// TIA Portal V16 program export: 1 tag tables, 16 data types, 7 data blocks, 22 code blocks (in call order from the OBs), 5 instance data blocks

VAR_GLOBAL   // PLC tag table "Default tag table"
   System_Byte AT %MB1 : Byte;
   FirstScan AT %M1.0 : Bool;
   DiagStatusUpdate AT %M1.1 : Bool;
   AlwaysTRUE AT %M1.2 : Bool;
   AlwaysFALSE AT %M1.3 : Bool;
   Clock_Byte AT %MB0 : Byte;
   Clock_10Hz AT %M0.0 : Bool;
   Clock_5Hz AT %M0.1 : Bool;
   "Clock_2.5Hz" AT %M0.2 : Bool;
   Clock_2Hz AT %M0.3 : Bool;
   "Clock_1.25Hz" AT %M0.4 : Bool;
   Clock_1Hz AT %M0.5 : Bool;
   "Clock_0.625Hz" AT %M0.6 : Bool;
   "Clock_0.5Hz" AT %M0.7 : Bool;
   ala AT %MW2 : Int;
   "di24.2" AT %I0.2 : Bool;
   diSAFETY AT %I0.3 : Bool;
   diC201FC01 AT %I0.4 : Bool;
   diC202FC01 AT %I0.5 : Bool;
   diC202AV03c AT %I0.6 : Bool;
   diC202AV04c AT %I0.7 : Bool;
   diC201AV01c AT %I1.0 : Bool;
   diC201AV02c AT %I1.1 : Bool;
   diC202AV01c AT %I1.2 : Bool;
   diC202AV02c AT %I1.3 : Bool;
   diC211AV01c AT %I1.4 : Bool;
   diC212AV01c AT %I1.5 : Bool;
   diC2A1AV01c AT %I1.6 : Bool;
   diC2A1AV02c AT %I1.7 : Bool;
   diC2A1AV11c AT %I2.0 : Bool;
   diC2A1AV12c AT %I2.1 : Bool;
   diC2A1AV31c AT %I2.2 : Bool;
   diC2A1AV41c AT %I2.3 : Bool;
   diC2D1AV01c AT %I2.4 : Bool;
   diC2D1AV11c AT %I2.5 : Bool;
   diC2D1AV41c AT %I2.6 : Bool;
   diC2D1AV42c AT %I2.7 : Bool;
   diC2D2AV01c AT %I3.0 : Bool;
   diC2D2AV11c AT %I3.1 : Bool;
   diC2D2AV41c AT %I3.2 : Bool;
   diC2D2AV42c AT %I3.3 : Bool;
   diC2D3AV01c AT %I3.4 : Bool;
   diC2D3AV11c AT %I3.5 : Bool;
   diC2D3AV31c AT %I3.6 : Bool;
   diC2D3AV41c AT %I3.7 : Bool;
   diC2D3AV42c AT %I4.0 : Bool;
   diC2D3AV43c AT %I4.1 : Bool;
   diC2L1AV01c AT %I4.2 : Bool;
   diC2L1AV02c AT %I4.3 : Bool;
   diC2L1AV11c AT %I4.4 : Bool;
   diC2L1AV12c AT %I4.5 : Bool;
   diC2L1AV31c AT %I4.6 : Bool;
   diC2L1AV41c AT %I4.7 : Bool;
   diC2R1AV01c AT %I5.0 : Bool;
   diC2R1AV02c AT %I5.1 : Bool;
   diC2R1AV11c AT %I5.2 : Bool;
   diC2R1AV12c AT %I5.3 : Bool;
   diC2R1AV41c AT %I5.4 : Bool;
   diC2W1AV02c AT %I5.5 : Bool;
   diC2W1AV31c AT %I5.6 : Bool;
   diC2W1AV41c AT %I5.7 : Bool;
   diC211FV01 AT %I6.0 : Bool;
   diC212FV01 AT %I6.1 : Bool;
   diC2D1FV81 AT %I6.2 : Bool;
   diC2D2FV81 AT %I6.3 : Bool;
   diC2A1PD01 AT %I6.4 : Bool;
   diC2D1PD01 AT %I6.5 : Bool;
   diC2D2PD01 AT %I6.6 : Bool;
   diC2D3PD01 AT %I6.7 : Bool;
   diC2L1PD01 AT %I7.0 : Bool;
   diC2R1PD01 AT %I7.1 : Bool;
   diC2W1PD01 AT %I7.2 : Bool;
   diC2A1LL01 AT %I7.3 : Bool;
   diC2D1LL01 AT %I7.4 : Bool;
   diC2D2LL01 AT %I7.5 : Bool;
   diC2D3LL01 AT %I7.6 : Bool;
   diC2L1LL01 AT %I7.7 : Bool;
   diC2R1LL01 AT %I8.0 : Bool;
   diC2W1LL01 AT %I8.1 : Bool;
   diC2A1LH01 AT %I8.2 : Bool;
   diC2D1LH01 AT %I8.3 : Bool;
   diC2D2LH01 AT %I8.4 : Bool;
   diC2D3LH01 AT %I8.5 : Bool;
   diC2L1LH01 AT %I8.6 : Bool;
   diC2R1LH01 AT %I8.7 : Bool;
   diC2W1LH01 AT %I9.0 : Bool;
   doC201AV21b AT %Q0.0 : Bool;
   doC202AV21b AT %Q0.1 : Bool;
   doC2W1AV31b AT %Q0.2 : Bool;
   doC2W1AV02b AT %Q0.3 : Bool;
   doC2R1AV11b AT %Q0.4 : Bool;
   doC2R1AV12b AT %Q0.5 : Bool;
   doC2R1AV41b AT %Q0.6 : Bool;
   doC2R1AV01b AT %Q0.7 : Bool;
   doC2R1AV02b AT %Q1.0 : Bool;
   doC2L1AV11b AT %Q1.1 : Bool;
   doC2L1AV12b AT %Q1.2 : Bool;
   doC2L1AV41b AT %Q1.3 : Bool;
   doC2L1AV01b AT %Q1.4 : Bool;
   doC2L1AV02b AT %Q1.5 : Bool;
   doC2L1AV31b AT %Q1.6 : Bool;
   doC2A1AV11b AT %Q1.7 : Bool;
   doC2A1AV12b AT %Q2.0 : Bool;
   doC2A1AV41b AT %Q2.1 : Bool;
   doC2A1AV01b AT %Q2.2 : Bool;
   doC2A1AV02b AT %Q2.3 : Bool;
   doC2A1AV31b AT %Q2.4 : Bool;
   doC2D1AV11b AT %Q2.5 : Bool;
   doC2D1AV41b AT %Q2.6 : Bool;
   doC2D1AV42b AT %Q2.7 : Bool;
   doC2D1AV01b AT %Q3.0 : Bool;
   doC2D2AV01b AT %Q3.1 : Bool;
   doC2D2AV42b AT %Q3.2 : Bool;
   doC2D2AV41b AT %Q3.3 : Bool;
   doC2D2AV11b AT %Q3.4 : Bool;
   doC2D3AV41b AT %Q3.5 : Bool;
   doC2D3AV42b AT %Q3.6 : Bool;
   doC2D3AV11b AT %Q3.7 : Bool;
   doC2D3AV31b AT %Q4.0 : Bool;
   doC2D3AV43b AT %Q4.1 : Bool;
   doC2D3AV01b AT %Q4.2 : Bool;
   doC202AV01b AT %Q4.3 : Bool;
   doC202AV02b AT %Q4.4 : Bool;
   doC201AV01b AT %Q4.5 : Bool;
   doC201AV02b AT %Q4.6 : Bool;
   doC2A1AV42b AT %Q5.0 : Bool;
   doC2L1AV42b AT %Q5.1 : Bool;
   doC2D1AV81b AT %Q5.3 : Bool;
   doC2D2AV81b AT %Q5.4 : Bool;
   doC2W1AV41b AT %Q5.5 : Bool;
   doC211AV01b AT %Q5.6 : Bool;
   doC212AV01b AT %Q5.7 : Bool;
   doC202AV03b AT %Q6.0 : Bool;
   doC202AV04b AT %Q6.1 : Bool;
   doC2A1MP41b AT %Q6.6 : Bool;
   doC2L1MP41b AT %Q6.7 : Bool;
   doBuczek AT %Q7.0 : Bool;
   doZielona AT %Q7.1 : Bool;
   doCzerwona AT %Q7.2 : Bool;
   doZolta AT %Q7.3 : Bool;
   aiC2W1TT01 AT %IW10 : Int;
   aiC2R1TT01 AT %IW12 : Int;
   aiC2L1TT01 AT %IW14 : Int;
   aiC2A1TT01 AT %IW16 : Int;
   aiC2D1TT01 AT %IW18 : Int;
   aiC2D2TT01 AT %IW20 : Int;
   aiC2D3TT01 AT %IW22 : Int;
   aiC211TT01 AT %IW24 : Int;
   aiC212TT01 AT %IW26 : Int;
   aiC201TT01 AT %IW28 : Int;
   aiC202TT01 AT %IW30 : Int;
   aiC212QIC01 AT %IW32 : Int;
   aiC211QIC01 AT %IW34 : Int;
   aiC2A1LT01 AT %IW36 : Int;
   aiC2D1LT01 AT %IW38 : Int;
   aiC2D2LT01 AT %IW40 : Int;
   aiC2D3LT01 AT %IW42 : Int;
   aiC2L1LT01 AT %IW44 : Int;
   aiC2R1LT01 AT %IW46 : Int;
   aiC2W1LT01 AT %IW48 : Int;
   aoC201CV21 AT %QW8 : Int;
   aoC202CV21 AT %QW10 : Int;
   aoC201FC01 AT %QW12 : Int;
   aoC202FC01 AT %QW14 : Int;
   aoC2D1MP81 AT %QW16 : Int;
   aoC2D2MP81 AT %QW18 : Int;
   C202FT01volume AT %ID50 : Real;
   C201FT01volume AT %ID85 : Real;
   C202FT01temperature AT %ID120 : Real;
   C201FT01temperature AT %ID125 : Real;
   doC2A1AV43b AT %Q4.7 : Bool;
   doC2L1AV43b AT %Q5.2 : Bool;
   "di24.1" AT %I0.1 : Bool;
   C2L1MP41 AT %MW10 : Int;
   C2A1AV01 AT %MW94 : Int;
   C202AV01 AT %MW80 : Int;
   C2A1MP41 AT %MW8 : Int;
   C2A1AV41 AT %MW104 : Int;
   C2D1FV81 AT %MW70 : Int;
   C2W1LL01 AT %MW62 : Int;
   C2D1PD01 AT %MW30 : Int;
   C2R1LL01 AT %MW56 : Int;
   C2D3PD01 AT %MW44 : Int;
   C2D3LL01 AT %MW42 : Int;
   C2L1AV43 AT %MW110 : Int;
   C201AV21 AT %MW78 : Int;
   C2A1PD01 AT %MW22 : Int;
   C2W1PD01 AT %MW64 : Int;
   C2D2FV81 AT %MW72 : Int;
   C202AV02 AT %MW82 : Int;
   C211AV01 AT %MW90 : Int;
   C2L1LH01 AT %MW46 : Int;
   C2D2LH01 AT %MW32 : Int;
   C2D1AV01 AT %MW112 : Int;
   diC2D2LL81 AT %I9.4 : Bool;
   C202AV21 AT %MW88 : Int;
   C2L1Ll41 AT %MW50 : Int;
   C212AV01 AT %MW92 : Int;
   C2A1AV12 AT %MW100 : Int;
   C211FV01 AT %MW66 : Int;
   C2R1PD01 AT %MW58 : Int;
   C2A1AV42 AT %MW106 : Int;
   diC2D1LL81 AT %I9.3 : Bool;
   C202FC01 AT %MW4 : Int;
   C2L1Ll01 AT %MW48 : Int;
   diC2A1LL41 AT %I9.1 : Bool;
   diC2L1LL41 AT %I9.2 : Bool;
   C2A1LH01 AT %MW16 : Int;
   C202AV03 AT %MW84 : Int;
   C2D2MP81 AT %MW14 : Int;
   C2D2LL01 AT %MW34 : Int;
   C2L1PD01 AT %MW52 : Int;
   C2D1LL81 AT %MW28 : Int;
   C2W1LH01 AT %MW60 : Int;
   C2A1AV02 AT %MW96 : Int;
   C2R1LH01 AT %MW54 : Int;
   C201AV01 AT %MW74 : Int;
   C2D1LH01 AT %MW24 : Int;
   C2D1LL01 AT %MW26 : Int;
   C2A1LL41 AT %MW20 : Int;
   C202AV04 AT %MW86 : Int;
   C212FV01 AT %MW68 : Int;
   C2D1MP81 AT %MW12 : Int;
   C2A1LL01 AT %MW18 : Int;
   C2A1AV31 AT %MW102 : Int;
   C2D2PD01 AT %MW38 : Int;
   C201AV02 AT %MW76 : Int;
   C2D3LH01 AT %MW40 : Int;
   C2D2LL81 AT %MW36 : Int;
   C2A1AV11 AT %MW98 : Int;
   C2A1AV43 AT %MW108 : Int;
   C2D1AV41 AT %MW116 : Int;
   C2L1AV31 AT %MW152 : Int;
   C2L1AV41 AT %MW154 : Int;
   C2R1AV12 AT %MW164 : Int;
   C211QIC01 AT %MW218 : Int;
   CD1LT01 AT %MW198 : Int;
   C2D3AV11 AT %MW134 : Int;
   C2L1AV01 AT %MW144 : Int;
   C2L1AV12 AT %MW150 : Int;
   C2L1AV11 AT %MW148 : Int;
   C2D3TT01 AT %MW186 : Int;
   CD2LT01 AT %MW200 : Int;
   C2D1AV81 AT %MW120 : Int;
   C2D1TT01 AT %MW182 : Int;
   C201CV21 AT %MW220 : Int;
   C2L1LT01 AT %MW210 : Int;
   C2D3AV42 AT %MW140 : Int;
   C211TT01 AT %MW188 : Int;
   C2D2AV41 AT %MW126 : Int;
   C2D2AV01 AT %MW122 : Int;
   C2D2LT01 AT %MW204 : Int;
   C2D3AV01 AT %MW132 : Int;
   C2W1LT01 AT %MW214 : Int;
   CD3LT01 AT %MW202 : Int;
   C2D2AV42 AT %MW128 : Int;
   C2R1LT01 AT %MW212 : Int;
   C2D2TT01 AT %MW184 : Int;
   C2A1LT01 AT %MW196 : Int;
   C202TT01 AT %MW194 : Int;
   C2L1TT01 AT %MW178 : Int;
   C2R1AV01 AT %MW158 : Int;
   C2D1LT01 AT %MW208 : Int;
   C212TT01 AT %MW190 : Int;
   C212QIC01 AT %MW216 : Int;
   C2D2AV11 AT %MW124 : Int;
   C201TT01 AT %MW192 : Int;
   C2D3AV31 AT %MW136 : Int;
   C2D3LT01 AT %MW206 : Int;
   C2RW1AV31 AT %MW170 : Int;
   C2A1TT01 AT %MW180 : Int;
   C202CV21 AT %MW222 : Int;
   C2R1AV11 AT %MW162 : Int;
   C2RW1AV02 AT %MW168 : Int;
   C2D3AV41 AT %MW138 : Int;
   C2L1AV02 AT %MW146 : Int;
   C2R1TT01 AT %MW176 : Int;
   C2R1AV41 AT %MW166 : Int;
   C2RW1AV41 AT %MW172 : Int;
   C2D1AV42 AT %MW118 : Int;
   C2W1TT01 AT %MW174 : Int;
   C2R1AV02 AT %MW160 : Int;
   C2D2AV81 AT %MW130 : Int;
   C2D3AV43 AT %MW142 : Int;
   C2D1AV11 AT %MW114 : Int;
   C2L1AV42 AT %MW156 : Int;
   staryNumerObiektuWybranyZHMI AT %MW226 : Int;
   numerObiektuWybranyZHMI AT %MW224 : Int;
   doC2W1AV01b AT %Q7.4 : Bool;
   C2W1AV01 AT %MW228 : Int;
   diC2W1AV01c AT %I9.7 : Bool;
   C2W1AV02 AT %MW230 : Int;
   doC2D2MP81 AT %Q6.3 : Bool;
   doC202FC01 AT %Q6.5 : Bool;
   doC2D1MP81 AT %Q6.2 : Bool;
   doC201FC01 AT %Q6.4 : Bool;
   hmi_alarm AT %M232.0 : Bool;
   C2W1AV41 AT %MW236 : Int;
   C2W1AV31 AT %MW234 : Int;
   "Cip1.pompaPodawaniaCip" AT %MW6 : Int;
   linia1_pompa_zezwolenie AT %M232.1 : Bool;
   krokZapauzowany AT %MW238 : Int;
   numer_kroku_stary_1 AT %MW240 : Int;
   numer_kroku_stary_2 AT %MW242 : Int;
END_VAR
VAR_GLOBAL CONSTANT   // user constants
   f101fc01 : Int := 2;
END_VAR

TYPE "typAlarmNew"
// stored: IsFailsafeCompliant false
   STRUCT
      stan : Int;   // 0-bark 1-wystapił i jest alarm
      procedura { ExternalAccessible := 'False'; ExternalVisible := 'False'; ExternalWritable := 'False'} : Int;   // numer procedury któa teraz wykonujemy
      timerek { ExternalAccessible := 'False'; ExternalVisible := 'False'; ExternalWritable := 'False'} : Int;   // czas liczony do wystapienia alarmu
   END_STRUCT;
END_TYPE

TYPE "typButton"
// stored: IsFailsafeCompliant false
   STRUCT
      set : Bool;
      reset : Bool;
      widoczny : Bool := 1;
      kolor : Int := 4;
      aktywny : Bool := 1;
   END_STRUCT;
END_TYPE

TYPE "typFlipaj"
// stored: IsFailsafeCompliant false
   STRUCT
      in { ExternalAccessible := 'False'; ExternalVisible := 'False'; ExternalWritable := 'False'} : Bool;
      start_od_zera { ExternalAccessible := 'False'; ExternalVisible := 'False'; ExternalWritable := 'False'} : Bool;   // że po wyzwoleniu jest najpierw OFF
      Q { ExternalAccessible := 'False'; ExternalVisible := 'False'; ExternalWritable := 'False'} : Bool;
      ile_petli { ExternalAccessible := 'False'; ExternalVisible := 'False'; ExternalWritable := 'False'} : Int;   // że filpanie ma dziać się w kółko
      czas_ON { ExternalAccessible := 'False'; ExternalVisible := 'False'; ExternalWritable := 'False'} : Int;   // czas załączenia wyjścia 0.1 s
      czas_OFF { ExternalAccessible := 'False'; ExternalVisible := 'False'; ExternalWritable := 'False'} : Int;   // czas wyłączenia wyjścia 0.1s
      licznik_petli { ExternalAccessible := 'False'; ExternalVisible := 'False'; ExternalWritable := 'False'} : Int;
      licznik { ExternalAccessible := 'False'; ExternalVisible := 'False'; ExternalWritable := 'False'} : LInt;
   END_STRUCT;
END_TYPE

TYPE "typFunkcjeObiektówCipu"
// stored: IsFailsafeCompliant false
   STRUCT
      "-na stacji CIP duże zbiorniki i zawory pod nimi" : Bool;   // tor0 to urządzenia wykorzystywane podczas pracy obu torów 1 i 2
      pompaPodawaniaCip : Int;   // najczęściej na torach 1 i 2
      zawórZrzutowyDoKanalizacji : Int;   // najczęściej na torach 1 i 2
      zawórWydawczyCip : Int;   // najczęściej na torach 1 i 2
      zawórBypassPrzygotowaniaStacji : Int;   // najczęściej na torach 1 i 2
      zawórParowyOdcinający : Int;   // najczęściej na torach 1 i 2
      zawórParowyRegulacyjny : Int;   // najczęściej na torach 1 i 2
      zawórWydawczyWodyWtórnej : Int;   // najczęściej na torach 1 i 2
      zawórPowrotnyWodyWtórnej : Int;   // najczęściej na torach 1 i 2
      zawórWydawczyŁugu : Int;   // najczęściej na torach 1 i 2
      zawórPowrotnyŁugu : Int;   // najczęściej na torach 1 i 2
      zawórWydawczyKwasu : Int;   // najczęściej na torach 1 i 2
      zawórPowrotnyKwasu : Int;   // najczęściej na torach 1 i 2
      zawórWydawczyWodyCzystej : Int;   // najczęściej na torach 1 i 2
      zawórWydawczyDezynfekantu : Int;   // najczęściej na torach 1 i 2 - patrz Orzeł2 2019_1109
      zawórWydawczyDezynfekantu_2 : Int;   // najczęściej na torach 1 i 2 - patrz Orzeł2 2019_1109
      zawórPowrotnyDezynfekantu : Int;   // najczęściej na torach 1 i 2 - patrz Orzeł2 2019_1109
      zawórPowrotnyDezynfekantu_2 : Int;   // najczęściej na torach 1 i 2 - patrz Orzeł2 2019_1109
      zawórStopowyPowrotuDezynfekantu : Int;   // najczęściej na torach 1 i 2 - patrz Orzeł2 2019_1109
      zawórStopowyPowrotuDezynfekantu_2 : Int;   // najczęściej na torach 1 i 2 - patrz Orzeł2 2019_1109
      zawórNaGruszkęZbiornikaŁugu : Int;   // najczęściej na torze 1 lub na torze 2 (mycie się stacji)
      zawórNaGruszkęZbiornikaKwasu : Int;   // najczęściej na torze 1 lub na torze 2 (mycie się stacji)
      zawórNaGruszkęZbiornikaWodyWtórnej : Int;   // najczęściej na torze 1 lub na torze 2 (mycie się stacji)
      zawórNaGruszkęZbiornikaWodyCzystej : Int;   // najczęściej na torze 1 lub na torze 2 (mycie się stacji)
      zawórNaGruszkęZbiornikaDezynfekantu : Int;   // najczęściej na torach 1 i 2 - patrz Orzeł2 2019_1109
      zawórNaGruszkęZbiornikaDezynfekantu_2 : Int;   // najczęściej na torach 1 i 2 - patrz Orzeł2 2019_1109
      zawórWodaNaGruszkęZbiornikaDezynfekantu_2 : Int;   // najczęściej na torach 1 i 2 - patrz Orzeł2 2019_1109
      zawórUzupełnianiaWodyCzystejZbŁugu : Int;   // najczęsciej tor 0
      zawórUzupełnianiaWodyCzystejZbKwasu : Int;   // najczęsciej tor 0
      zawórUzupełnianiaWodyCzystejZbWodyWtórnej : Int;   // najczęsciej tor 0
      zawórUzupełnianiaWodyCzystejZbWodyCzystej : Int;   // najczęsciej tor 0
      ZawórUzupełnianiaWodyCzystejZbDezynfekantu : Int;   // najczęsciej tor 0
      ZawórUzupełnianiaWodyCzystejZbDezynfekantu_2 : Int;   // najczęsciej tor 0
      "---zbiorniki główne na stacji CIP -czujniki" : Bool;
      zbiornikŁugu : Struct
         czujnikDolnegoPoziomu : Int;
         czujnikGórnegoPoziomu : Int;
         temperatura : Int;
         poziomAnalogowy : Int;
         czujnikwłazu : Int;
      END_STRUCT;
      zbiornikKwasu : Struct
         czujnikDolnegoPoziomu : Int;
         czujnikGórnegoPoziomu : Int;
         temperatura : Int;
         poziomAnalogowy : Int;
         czujnikwłazu : Int;
      END_STRUCT;
      zbiornikWodyWtórnej : Struct
         czujnikDolnegoPoziomu : Int;
         czujnikGórnegoPoziomu : Int;
         temperatura : Int;
         poziomAnalogowy : Int;
         czujnikwłazu : Int;
      END_STRUCT;
      zbiornikwodyCzystej : Struct
         czujnikDolnegoPoziomu : Int;
         czujnikGórnegoPoziomu : Int;
         temperatura : Int;
         poziomAnalogowy : Int;
         czujnikwłazu : Int;
      END_STRUCT;
      zbiornikDezynfekantu : Struct
         czujnikDolnegoPoziomu : Int;
         czujnikGórnegoPoziomu : Int;
         temperatura : Int;
         poziomAnalogowy : Int;
         czujnikwłazu : Int;
         zbiornikDezynfekantu : Struct
            czujnikDolnegoPoziomu : Int;
            czujnikGórnegoPoziomu : Int;
            temperatura : Int;
            poziomAnalogowy : Int;
            czujnikwłazu : Int;
         END_STRUCT;
      END_STRUCT;
      zbiornikDezynfekantu_2 : Struct
         czujnikDolnegoPoziomu : Int;
         czujnikGórnegoPoziomu : Int;
         temperatura : Int;
         poziomAnalogowy : Int;
         czujnikwłazu : Int;
      END_STRUCT;
      "-zbiorniki na stacji przygotowania chemii" : Bool;
      zbiorniczekDozowaniaŁugu : Struct   // na stacji przygotowania chemii
         czujnikDolnegoPoziomu : Int;
         czujnikGórnegoPoziomu : Int;
         temperatura : Int;
         poziomAnalogowy : Int;
         czujnikwłazu : Int;
         zbiornikDezynfekantu : Struct
            czujnikDolnegoPoziomu : Int;
            czujnikGórnegoPoziomu : Int;
            temperatura : Int;
            poziomAnalogowy : Int;
            czujnikwłazu : Int;
         END_STRUCT;
      END_STRUCT;
      zbiorniczekDozowaniaKwasu : Struct   // na stacji przygotowania chemii
         czujnikDolnegoPoziomu : Int;
         czujnikGórnegoPoziomu : Int;
         temperatura : Int;
         poziomAnalogowy : Int;
         czujnikwłazu : Int;
         zbiornikDezynfekantu : Struct
            czujnikDolnegoPoziomu : Int;
            czujnikGórnegoPoziomu : Int;
            temperatura : Int;
            poziomAnalogowy : Int;
            czujnikwłazu : Int;
         END_STRUCT;
      END_STRUCT;
      zbiorniczekDozowanieDezynfekantu : Struct   // na stacji przygotowania chemii
         czujnikDolnegoPoziomu : Int;
         czujnikGórnegoPoziomu : Int;
         temperatura : Int;
         poziomAnalogowy : Int;
         czujnikwłazu : Int;
         zbiornikDezynfekantu : Struct
            czujnikDolnegoPoziomu : Int;
            czujnikGórnegoPoziomu : Int;
            temperatura : Int;
            poziomAnalogowy : Int;
            czujnikwłazu : Int;
         END_STRUCT;
      END_STRUCT;
      "--nalinii" : Bool;
      temperaturaZaWymiennikiem : Int;   // najczęściej na torach 1 i 2
      przepływomierzZaWymiennikiem : Int;   // najczęściej na torach 1 i 2
      temperaturaNaPowrocie : Int;   // najczęściej na torach 1 i 2
      przewodnośćNaPowrocie : Int;   // najczęściej na torach 1 i 2
      czujnikPrzepływuNaPowrocie : Int;   // najczęściej na torach 1 i 2
      "-naobiekcie" : Bool;
      czujnikDolnegoPoziomuwZbiornikuDrenowanym : Int;   // najczęściej na torach 1 i 2 (sygnał z obiektu mytego)
      "-przygotowaniechemii" : Bool;
      pompkaDozowaniaŁuguwLinię : Int;   // najczęsciej tor 0
      pompkaDozowaniaKwasuwLinię : Int;   // najczęsciej tor 0
      pompkaDozowaniaDezynfekantuwLinię : Int;   // najczęściej na torach 1 i 2
      zawórDozowaniaLuguwLinię : Int;   // najczęściej na torach 1 i 2
      zawórDozowaniaKwasuwLinię : Int;   // najczęściej na torach 1 i 2
      zawórDozowaniaDezynfekantuwLinię : Int;   // najczęściej na torach 1 i 2
      czujnikPrzepływuDozowanegoŁugu : Int;   // najczęsciej tor 0
      czujnikPrzepływuDozowanegoKwasu : Int;   // najczęsciej tor 0
      czujnikPrzepływuDozowanegoDezynfekantu : Int;   // najczęściej na torach 1 i 2
      PrzepływomierzDozowanejChemii : Int;   // najczęsciej tor 0
   END_STRUCT;
END_TYPE

TYPE "typKlawiszeProdukcji"
// stored: IsFailsafeCompliant false
   STRUCT
      bStart { S7_SetPoint := 'True'} : "typButton";   // Aktywacja podświetla klawisz na zielono (Start pali się zawsze z innymi klawiszami)
      bPauza { S7_SetPoint := 'True'} : "typButton";   // Przytrzymanie Klawisza aktywuje K6700 (program musi pamiętać z jakiego kroku wyszedł/do jakiego ma wrócić)
      bStop { S7_SetPoint := 'True'} : "typButton";   // Przytrzymanie przez 5s K6100
      bProdukcja { S7_SetPoint := 'True'} : "typButton";   // aktywacja podświetla klawisz na zielono
      bCyrkulacja { S7_SetPoint := 'True'} : "typButton";   // aktywacja podświetla klawisz na żółto; awaryjnie na czerwono
      bCip { S7_SetPoint := 'True'} : "typButton";   // aktywacja podświetla klawisz na zielono
      bPullout { S7_SetPoint := 'True'} : "typButton";   // aktywacja podświetla klawisz na zielono
      bFlux { S7_SetPoint := 'True'} : "typButton";
      bNastepnyKrok { S7_SetPoint := 'True'} : "typButton";   // nastepny krok wyskakuje podczas mycia jezeli alarm 18
      bPrzygotowanie { S7_SetPoint := 'True'} : "typButton";   // przygotowanie stacji CIP
   END_STRUCT;
END_TYPE

TYPE "typKrokRecepturyStacjiMycia"
// stored: IsFailsafeCompliant false
   STRUCT
      nazwaKroku : WString[33] := WSTRING#'nazwa receptury';   // nazwa kroku
      PM : Array[0..30] of Real;
   END_STRUCT;
   // // PM[1] : krokAktywny
   // // PM[2] : wydajnośćMycia
   // // PM[3] : czasOczekiwaniaNaZasilanie
   // // PM[4] : CzasOczekiwaniaNaPowrót
   // // PM[5] : ObjętośćPłukania
   // // PM[6] : CzasMycia
   // // PM[7] : CzasOdsączania
   // // PM[8] : Objetość WypełnieniaDoGruszki
   // // PM[9] : CzasOpóżnieniaUruchomieniaPompyCIP
   // // PM[10] : StężeniaMinimalne
   // // PM[11] : StężenieDozowania
   // // PM[12] : StężeniePłukania
   // // PM[13] : TemperaturaProcesu
   // // PM[14] : TemperaturaPłukania
   // // PM[15] : HisterezaStężeniaDoRozpoczęciaOdliczania
   // // PM[16] : RóznicaTemperaturDoRozpoczęciaOdliczania
   // // PM[17] : WspółczynnikKompensacji
   // // PM[18] : TemperaturaOdniesieniaKompensacji
   // // PM[19] : MaksymalnyCzasOperacji
   // // PM[20] : CzasDozowaniaChemii
   // // PM[21] : SprawdzanieCzujników
   // // PM[22] : KompensacjaTemperaturowa
   // // PM[23] : MycieTanku
   // // PM[24] : CIPsp201 optymalizacja objetosci
   // // PM[25] : Cipsp202 optymalizacja stezen
   // // PM[26] : czas załączenia pompki chemii
   // // PM[27] : czas wyłączenia pompki chemii
END_TYPE

TYPE "typObiekt"
// stored: IsFailsafeCompliant false
   STRUCT
      typObiektu : Int := 1;
      nazwaObiektu : String[10] := 'F100AV01';
      procedura : Int;   // procedura 0 - to wyłaczenie/procedura 1 to załączenie
      inStartAuto : Bool;
      outStartUrządzenie : Bool;
      inLiftUp : Bool;
      outLiftUp : Bool;
      inLiftDown : Bool;
      outLiftDown : Bool;
      inZadaneWysterowanieAuto : Real;
      outWysterowanieUrządzenia : Real;
      inJestPotwWysterowania : Bool;
      diPotwWysterowania : Bool;
      inJestPotwNiewysterowania : Bool;
      diPotwNieWysterowania : Bool;
      inZezwolenieNaPracę : Bool;   // pkz+KSB+CKF+przełacznik wyłacznika siremontowego / z KSB
      Awaria : Bool;   // bit informujacy o awarii
      ResetAwaria : Bool;   // reset z programu
      kodBłedu : Word;   // kod statusu z urządzenia (falownik słowo statusu)
      czasDoAwariiSP : Int := 1000;
      czasDoAwariiPV : Int;
      czasPracyGodziny : Real;   // np. czas pracy pompy
      _ : Bool;
      hmiPokażStacyjkę : Bool;   // //stacyjka
      hmiStanUrządzenia : Int;   // rysunek na hmi
      hmiTrybAutoManual : Bool;   // zmiana trybu pracy urządzenia ze stacyjki
      hmiManualStart : Bool;   // /maualne załączenie pompy zaworu
      hmiManualStop : Bool;   // tylko żeby w stacujce pokazac przycisk/lampke
      hmiManualLiftUp : Bool;   // dla zaworów
      hmiManualLiftDown : Bool;   // dla zaworów
      hmiManualneWysterowanie : Real;   // /manualna wartosc analogowa ręka pompy /pida
      hmiSymulujSygnałyWejsciowe : Bool;   // załącz maskowanie/symulacje wejsc
      hmiSymulacjaPotwWysterowania : Bool;
      hmiSymulacjaPotwNieWysterowania : Bool;
      hmiSymulowanaWartośćAnalogowa : Real;   // symulowana wartość pomiarowa dla mierników
      hmiPotwNieWysterowania : Bool;
      hmiPotwWysterowania : Bool;   // wynikowy bit potwierdzenia wysterowania
      hmiZasilanieOK : Bool;   // potwierdzenie że termik załaczoony/ zasilanie falownika ok
      hmiResetAwaria : Bool;   // reset ze stacyjki
      hmiPrądFalownika : Real;   // prad falownika
      ___ : Bool;   // ////////////////////analogi///////////////////////
      inPomiarRaw : Int;   // wejście ai sterownika (0-27648) / pomiar
      minSkali : Real := -50.0;   // wartość dla 4mA - raw=0
      maxskali : Real := 150.0;   // wartość dla 20mA - raw 27648
      tFiltr : Real := 0.9;   // 0.8 -0.99 /d /rampa dla pompy 0 -99sekund
      pomiarTymczas : Real;
      wyjTymczas : Real;
      WartośćPomiaru : Real;   // pomiar analogowy
      ____ { ExternalWritable := 'False'} : Bool;   // ///////////////przepływomierz//////////////////////
      hmiMetry3NaImpuls : Real := 0.001;   // wartość nastawy dla wejścia impulsowego(jeżeli stosujemy)
      diImpulsy : Bool;   // wejście impulsowe z przepływomierza lub z programu
      R_Trig : Bool;   // impulsator z programu podczas załaczenia symulacji
      startLicznik1 : Bool;
      zerujLicznik1 : Bool;
      startLicznik2 : Bool;
      zerujLicznik2 : Bool;
      startLicznik3 : Bool;
      zerujLicznik3 : Bool;
      licznik1 : Real;
      licznik2 : Real;
      licznik3 : Real;
      licznikTotalImpulsy : Int;
      Lreal_1 : LReal;
      Lreal_2 : LReal;
      _____ : Bool;
      pid_SP : Real;   // //PID setpoint
      pid_PV : Real;   // proces value
      pid_P : Real := 1.0;
      pid_I : Real := 10.0;
      pid_D : Real;
      pid_Rampa : Real := 1.0;   // 0.0-1.0
      pid_Out : Real;
      ______ : Bool;
      SetReset { S7_SetPoint := 'True'} : "typSetReset";
      Flipaj : "typFlipaj";
      I1 { S7_SetPoint := 'True'} : Int;
      l2 : LReal;
      l4 : Word;
   END_STRUCT;
END_TYPE

TYPE "typProgram"
// stored: IsFailsafeCompliant false
   STRUCT
      nazwaFunkcji : Int;
      nazwaKroku : Int;
      numerKroku : Int;
      numerKrMycia : Int;
      zadana1 : Real;
      aktualna1 : Real;
      zadana2 : Real;
      aktualna2 : Real;
      opóżnienie : Real;
   END_STRUCT;
END_TYPE

TYPE "typRecepturaStacjiMycia"
// stored: IsFailsafeCompliant false
   STRUCT
      nazwaReceptury : WString[33] := WSTRING#'nazwa receptury';
      Krok { S7_SetPoint := 'True'} : Array[0..6] of "typKrokRecepturyStacjiMycia";
   END_STRUCT;
   // Krok[0].nazwaKroku := WSTRING#'';
   // Krok[1].nazwaKroku := WSTRING#'Płukanie Zimne';
   // Krok[2].nazwaKroku := WSTRING#'Płukanie Gorące';
   // Krok[3].nazwaKroku := WSTRING#'Ług';
   // Krok[4].nazwaKroku := WSTRING#'Kwas';
   // Krok[5].nazwaKroku := WSTRING#'Płukanie Główne';
   // Krok[6].nazwaKroku := WSTRING#'Dezynfekcja';
END_TYPE

TYPE "typSetReset"
// stored: IsFailsafeCompliant false
   STRUCT
      inSet : Bool;
      inReset : Bool;
      czasDoSet : Int;
      czasDoReset : Int;
      wyjście : Bool;
      setCzas : Int;
      resetCzas : Int;
   END_STRUCT;
END_TYPE

TYPE "typSygnałCiToObject"
// stored: IsFailsafeCompliant false
   STRUCT
      iCipLifeWord : UInt;   // lifeword:=lifeword+1 every 100ms
      iNrOfReqObjectToCip : UInt;   // Cip station tells you which object you want to clean
      iTimeToEndCip : UInt;   // remaining time to end of Cip process [seconds]
      bReqRouteToCip : Bool;   // Cip station request Object to set valves to Cip
      bCipIsActive : Bool;   // Cip statin informs of Active Cip process
      bReqPulloutTank : Bool;   // Cip station request Pullout process
      bReqStartReturnPump : Bool;   // Cip station request to start return pump (Cip-)
      bReqFlipValve : Bool;   // Cip station request Object ti flip valves
      bCipError : Bool;   // Cip station informs in Error
   END_STRUCT;
END_TYPE

TYPE "typSygnałONOFF"
// stored: IsFailsafeCompliant false
   STRUCT
      nazwaSygnału : String[10] := 'F100AV01';
      procedura : Int;   // procedura 0 - to wyłaczenie/procedura 1 to załączenie
      inStart : Bool;
      outStart : Bool;
      hmiTrybAutoManual : Bool;
      hmiManualStart : Bool;
      hmiStanUrządzenia : Int;
   END_STRUCT;
END_TYPE

TYPE "typSygnałObjectToCip"
// stored: IsFailsafeCompliant false
   STRUCT
      iLifeWord : UInt;   // lifeword:=lifeword+1 every 100ms
      iNrOfReadyObjectToCip : UInt;   // identification of ready object to Cip
      bReadyToCip : Bool;   // object is ready to Cip
      bTankisNotEmpty : Bool;   // show low-level sensor if tank is draining
      bReqPause : Bool;   // object request pause of Cip process
      bError : Bool;   // object send Error
   END_STRUCT;
END_TYPE

TYPE "typSygnałPomiędzyObiektamiMycia"
// stored: IsFailsafeCompliant false
   STRUCT
      toCip : "typSygnałObjectToCip";
      fromCip : "typSygnałCiToObject";
   END_STRUCT;
END_TYPE

TYPE "typSygnały"
// stored: IsFailsafeCompliant false
   STRUCT
      S : Array[1..50] of Bool;   // sygnał
   END_STRUCT;
   // // S[1] : CIP1
   // // S[2] : CIP2
   // // S[3] : CIP3
   // // S[4] : TANK_CIP
   // // S[5] : READY1
   // // S[6] : READY2
   // // S[7] : READY3
   // // S[8] : READY4
   // // S[9] : CONF1
   // // S[10] : CONF2
   // // S[11] : CONF3
   // // S[12] : CONF4
   // // S[13] : ERR
   // // S[14] : PULLOUT1
   // // S[15] : PULLOUT2
   // // S[16] : PULLOUT3
   // // S[17] : WATER1
   // // S[18] : WATER2
   // // S[19] : WATER3
   // // S[20] : OUT1
   // // S[21] : OUT2
   // // S[22] : OUT3
   // // S[23] : CONNECT1
   // // S[24] : CONNECT2
   // // S[25] : CONNECT3
   // // S[26] : WHEY
   // // S[27] : AG
   // // S[28] : PUMP
   // // S[29] : FLIP
   // // S[30] : RUNNING
   // // S[31] : FEED
   // // S[32] : START
   // // S[33] : REMOTE
   // // S[34] : RINSING
   // // S[35] : ERR
   // // S[36] : OUT
   // // S[37] : ZS01
   // // S[38] : ZS02
   // // S[39] : ZS03
   // // S[40] : ZS04
   // // S[41] : ZS05
END_TYPE

TYPE "typSygnałyzMaszyn"
// stored: IsFailsafeCompliant false
   STRUCT
      "M" : Array[1..5] of "typSygnały";   // maszyna
   END_STRUCT;
END_TYPE

DATA_BLOCK "CipSignals"   // DB1
{ S7_Optimized_Access := 'TRUE' }
VERSION : 0.1
// stored: AutoNumber true, DBAccessibleFromOPCUA true, IsOnlyStoredInLoadMemory false, IsRetainMemResEnabled false, IsWriteProtectedInAS false, MemoryReserve 100
   VAR
      Object : Array[0..20] of "typSygnałPomiędzyObiektamiMycia";
   END_VAR
BEGIN
END_DATA_BLOCK

DATA_BLOCK "DB_reports_mlekomat"   // DB12
{ S7_Optimized_Access := 'TRUE' }
VERSION : 0.1
// stored: AutoNumber true, DBAccessibleFromOPCUA true, IsOnlyStoredInLoadMemory false, IsRetainMemResEnabled false, IsWriteProtectedInAS false, MemoryReserve 100
   VAR RETAIN
      cips : Array[0..7] of Struct
         cip_active : Bool;   // teraz trwa mycie
         print_report : Bool;   // bit dla scady żeby wydrukowała raport
         print_report_done : Bool;   // bit ze skady ze raport się wydrukował
         number_of_cip : Int;   // aktualny numer kolejnego mycia w historii
         start_cip_date_and_time : Date_And_Time;
         start_lye_date_and_time : Date_And_Time;
         start_acid_date_and_time : Date_And_Time;
         start_disinfection_date_and_time : Date_And_Time;
         stop_cip_date_and_time : Date_And_Time;
      END_STRUCT;
   END_VAR
BEGIN
END_DATA_BLOCK

DATA_BLOCK "ms_na_procenty_DB"   // DB34
{ S7_Optimized_Access := 'TRUE' }
VERSION : 0.1
// blok danych dla funkcji ms_na_procenty
// stored: AutoNumber true, DBAccessibleFromOPCUA true, IsOnlyStoredInLoadMemory false, IsRetainMemResEnabled false, IsWriteProtectedInAS false, MemoryReserve 100
   VAR RETAIN
      inJednostkaAlkaliczna : Real;   // 1% środka alkalicznego= 48mS
      inJednostkaKwaśna : Real;   // 1% środka kwaśnego=56mS
      inPrzewodnośćCzystejWody { S7_SetPoint := 'True'} : Real;   // Przewodność czystej wody=0.3mS
   END_VAR
   VAR
      outStężenieŚrodkaTor1 : Real;
      outStężenieŚrodkaTor2 : Real;
   END_VAR
BEGIN
END_DATA_BLOCK

DATA_BLOCK "Tor1_hmi"   // DB2
{ S7_Optimized_Access := 'TRUE' }
VERSION : 0.1
// stored: AutoNumber true, DBAccessibleFromOPCUA true, IsOnlyStoredInLoadMemory false, IsRetainMemResEnabled false, IsWriteProtectedInAS false, MemoryReserve 100
   VAR
      button { S7_SetPoint := 'True'} : "typKlawiszeProdukcji";
      bPomińŁugowanie { S7_SetPoint := 'True'} : Bool;
      bPomińKwasowanie : Bool;
      bPomińDesynfekcje : Bool;
      bPomińPłukaniePoDezynfekcji : Bool;
   END_VAR
BEGIN
   button.bStart.widoczny := true;
END_DATA_BLOCK

DATA_BLOCK "Tor1_program"   // DB35
{ S7_Optimized_Access := 'TRUE' }
VERSION : 0.1
// stored: AutoNumber true, DBAccessibleFromOPCUA true, IsOnlyStoredInLoadMemory false, IsRetainMemResEnabled false, IsWriteProtectedInAS false, MemoryReserve 100
   VAR
      program : "typProgram";
   END_VAR
BEGIN
END_DATA_BLOCK

DATA_BLOCK "Tor2_hmi"   // DB3
{ S7_Optimized_Access := 'TRUE' }
VERSION : 0.1
// stored: AutoNumber true, DBAccessibleFromOPCUA true, IsOnlyStoredInLoadMemory false, IsRetainMemResEnabled false, IsWriteProtectedInAS false, MemoryReserve 100
   VAR
      button { S7_SetPoint := 'True'} : "typKlawiszeProdukcji";
      bPomińŁugowanie { S7_SetPoint := 'True'} : Bool;
      bPomińKwasowanie : Bool;
      bPomińDesynfekcje : Bool;
      bPomińPłukaniePoDezynfekcji : Bool;
   END_VAR
BEGIN
   button.bStart.widoczny := true;
END_DATA_BLOCK

DATA_BLOCK "Tor2_program"   // DB10
{ S7_Optimized_Access := 'TRUE' }
VERSION : 0.1
// stored: AutoNumber true, DBAccessibleFromOPCUA true, IsOnlyStoredInLoadMemory false, IsRetainMemResEnabled false, IsWriteProtectedInAS false, MemoryReserve 100
   VAR
      program : "typProgram";
   END_VAR
BEGIN
END_DATA_BLOCK

ORGANIZATION_BLOCK "Main"   // OB1, LAD, ProgramCycle
TITLE = "Main Program Sweep (Cycle)"
{ S7_Optimized_Access := 'TRUE' }
VERSION : 0.1
// stored: AutoNumber true, IsIECCheckEnabled false, SetENOAutomatically false
   VAR_INPUT
      Initial_Call : Bool;   // Initial call of this OB
      Remanence : Bool;   // =True, if remanent data are available
   END_VAR
BEGIN

REGION Network 1 (SCL)
   "ala" := "ala" + 1;
   "obsluga_stacyjki"();
END_REGION

REGION Network 2 (SCL)
   // #dlugosc := INT_TO_WORD(REAL_TO_INT("SIG".SIG[0]));//dlugosc paczki danych
   // //"liznik".liznik > 11 AND "liznik".liznik < 15
   // "BRCV_DB"(EN_R := (1),
   //           ID := W#16#116,
   //           R_ID := 3,
   //           STATUS => "status_reeed",
   //           RD_1 := "SIG".SIG,
   //           LEN := #dlugosc);
   // "R_TRIG_DB"(CLK := ("liznik".liznik >1 AND "liznik".liznik < 3));

   // "BSEND_DB"(REQ := ("R_TRIG_DB".Q),
   //            R := FALSE,
   //            ID := W#16#111,
   //            R_ID := 1,
   //            STATUS => "status_send",
   //            SD_1 := "SIG".SIG,
   //            LEN := #dlugosc);

   //     "PUT_DB"(REQ    := "Clock_10Hz",
   //              ID     := W#16#111,
   //              ADDR_1 := P#DB60.DBX0.0 int 1,
   //              SD_1   := P#DB23.DBX0.0 int 1);
END_REGION
END_ORGANIZATION_BLOCK

ORGANIZATION_BLOCK "100ms"
{ S7_Optimized_Access := 'TRUE' }
VERSION : 0.1

BEGIN
	//hw config - obsluga obiektow
	"Cip"();//obsluga obiektow
	"Cip.wejwyj"();//obsluga wej wyj
	
	//wywołanie programów 
	"Tor1.aMAIN"();
	"Tor2.aMAIN"();
	"Tor0.aMAIN"();
	
	
	// "hmi_alarm" := NOT "diSAFETY";//wykrzyknik na panelu hmi
	"hmi_alarm" := 0;
	
	
END_ORGANIZATION_BLOCK

FUNCTION "Cip.wejwyj" : Void
{ S7_Optimized_Access := 'TRUE' }
VERSION : 0.1
   VAR_TEMP 
      nr : Int;
      pomiar : Real;
      "bool" : Bool;
      "real" : Real;
      prąd : Real;
      częstotliwość : Real;
      diZasilanieOK : Bool;
      diKSB_OK : Bool;
      REALWEJSCIE : Real;
      aktualnyNumerReceptury : Int;
      aktualnyKrokMycia : Int;
   END_VAR


BEGIN
	// ;//tu przypisujemy nazwą obiektów ich numery  (np. "F101CP01" := 1;  -  zmienną F101CP01 typu integer deklaryjemy na początku programowania jako zmienną globalną
	// //w ten sposób okreslimy ilość obiektów i ich typy
	// //podpinamy wejscia wyjscia DO obiektów
	// // 
	
	#diKSB_OK := "diSAFETY";//kontrola przekażnika bezpieczeństwa
	#diZasilanieOK := "di24.1" AND "di24.2"; //napiecie z zasilaczy 24VDC
	#diKSB_OK := 1;
	#diZasilanieOK := 1;
	// /////////////////pompy na falowniku/regulowane
	// //
	#nr := 32;//tu wpisz nuemr obiektu
	"Cip".tor[1].pompaPodawaniaCip:= #nr; ;//tu przyporządkuj numer do obiektu na odpowiednim torze stacji
	"Cip".obiekt[#nr].nazwaObiektu := 'C201CP01';
	"Cip".obiekt[#nr].typObiektu := 4;
	"Cip".obiekt[#nr].inZezwolenieNaPracę := #diKSB_OK;
	"Cip".obiekt[#nr].hmiZasilanieOK := "diSAFETY";
	"Cip".obiekt[#nr].inJestPotwWysterowania := 1;
	"Cip".obiekt[#nr].diPotwWysterowania := "diC202FC01";
	"doC202FC01" := "Cip".obiekt[#nr].outStartUrządzenie;
	"aoC202FC01" := REAL_TO_INT("Cip".obiekt[#nr].outWysterowanieUrządzenia * 276.648);
	
	#nr := 31;//tu wpisz nuemr obiektu
	"C202FC01" := #nr;
	"Cip".tor[2].pompaPodawaniaCip := #nr; ;//tu przyporządkuj numer do obiektu na odpowiednim torze stacji
	"Cip".obiekt[#nr].nazwaObiektu := 'C202CP01';
	"Cip".obiekt[#nr].typObiektu := 4;
	"Cip".obiekt[#nr].inZezwolenieNaPracę := #diKSB_OK;
	"Cip".obiekt[#nr].hmiZasilanieOK := "diSAFETY";
	"Cip".obiekt[#nr].inJestPotwWysterowania := 1;
	"Cip".obiekt[#nr].diPotwWysterowania := "diC201FC01";
	"doC201FC01" := "Cip".obiekt[#nr].outStartUrządzenie;
	"aoC201FC01" := REAL_TO_INT("Cip".obiekt[#nr].outWysterowanieUrządzenia * 276.648);
	
	
	#nr := 97;//tu wpisz nuemr obiektu
	"C2D1MP81" := #nr;
	"Cip".tor[1].pompkaDozowaniaDezynfekantuwLinię := #nr; ;//tu przyporządkuj numer do obiektu na odpowiednim torze stacji
	"Cip".obiekt[#nr].nazwaObiektu := 'C2D1MP81';
	"Cip".obiekt[#nr].typObiektu := 4;
	"Cip".obiekt[#nr].inZezwolenieNaPracę := #diKSB_OK;
	"Cip".obiekt[#nr].hmiZasilanieOK := #diZasilanieOK;
	"Cip".obiekt[#nr].inJestPotwWysterowania := 1;
	"Cip".obiekt[#nr].diPotwWysterowania := "diC2D1FV81";
	"doC2D1MP81" := "Cip".obiekt[#nr].outStartUrządzenie;
	"aoC2D1MP81" := REAL_TO_INT("Cip".obiekt[#nr].outWysterowanieUrządzenia * 276.648);
	
	#nr := 98;//tu wpisz nuemr obiektu
	"C2D2MP81" := #nr;
	"Cip".tor[2].pompkaDozowaniaDezynfekantuwLinię:= #nr; ;//tu przyporządkuj numer do obiektu na odpowiednim torze stacji
	"Cip".obiekt[#nr].nazwaObiektu := 'C2D1MP81';
	"Cip".obiekt[#nr].typObiektu := 4;
	"Cip".obiekt[#nr].inZezwolenieNaPracę := #diKSB_OK;
	"Cip".obiekt[#nr].hmiZasilanieOK := #diZasilanieOK;
	"Cip".obiekt[#nr].inJestPotwWysterowania := 1;
	"Cip".obiekt[#nr].diPotwWysterowania := "diC2D2FV81";
	"doC2D2MP81" := "Cip".obiekt[#nr].outStartUrządzenie;
	"aoC2D2MP81" := REAL_TO_INT("Cip".obiekt[#nr].outWysterowanieUrządzenia * 276.648);
	
	
	
	//////////////////pompy on/off
	//
	#nr :=99;//tu wpisz nuemr obiektu
	"Cip".tor[0].pompkaDozowaniaKwasuwLinię := #nr; ;//tu przyporządkuj numer do obiektu na odpowiednim torze stacji
	"Cip".obiekt[#nr].nazwaObiektu := 'C2A1MP41';
	"Cip".obiekt[#nr].typObiektu := 3;
	"Cip".obiekt[#nr].hmiZasilanieOK := #diKSB_OK;
	"Cip".obiekt[#nr].inZezwolenieNaPracę := #diKSB_OK; ;
	"Cip".obiekt[#nr].inJestPotwWysterowania := 0;
	"Cip".obiekt[#nr].diPotwWysterowania :=0;
	"doC2A1MP41b" := "Cip".obiekt[#nr].outStartUrządzenie;
	
	// IF "Cip".obiekt["C2A1MP01"].hmiTrybAutoManual = 0 THEN
	//     "Cip".obiekt["C2A1MP01"].inStartAuto :=
	//     "Cip".obiekt["C2A1MP01"].inStartAuto
	//     OR "C22_obiekty".obiekt["C2A1MP01"].inStartAuto;
	//     "doC1A1MP01" := "Cip".obiekt["C2A1MP01"].inStartAuto;
	// END_IF;
	
	
	
	//
	#nr := 100;//tu wpisz nuemr obiektu
	"C2L1MP41" := #nr; ;//tu wpisz nazwę
	"Cip".tor[0].pompkaDozowaniaŁuguwLinię:= #nr; ;//tu przyporządkuj numer do obiektu na odpowiednim torze stacji
	"Cip".obiekt[#nr].nazwaObiektu := 'C2L1MP41';
	"Cip".obiekt[#nr].typObiektu := 3;
	"Cip".obiekt[#nr].hmiZasilanieOK := #diKSB_OK;
	"Cip".obiekt[#nr].inZezwolenieNaPracę := #diKSB_OK; ;
	"Cip".obiekt[#nr].inJestPotwWysterowania := 0;
	"Cip".obiekt[#nr].diPotwWysterowania := 0;
	"doC2L1MP41b" := "Cip".obiekt[#nr].outStartUrządzenie;
	
	
	// IF "Cip".obiekt["C2L1MP01"].hmiTrybAutoManual = 0 THEN
	//     "Cip".obiekt["C2L1MP01"].inStartAuto :=
	//     "Cip".obiekt["C2L1MP01"].inStartAuto
	//     OR "C22_obiekty".obiekt["C2L1MP01"].inStartAuto;
	//     "Cip".obiekt["C2L1MP01"].outStartUrządzenie := "Cip".obiekt["C2L1MP01"].inStartAuto;
	//     "doC1L1MP01" := "Cip".obiekt["C2L1MP01"].inStartAuto;
	// END_IF;
	
	
	
	// ///////////////////////////czujniki binarne ONOFF
	// //
	#nr := 42;//tu wpisz nuemr obiektu
	"Cip".tor[0].zbiornikKwasu.czujnikGórnegoPoziomu:= #nr; ;//tu przyporządkuj numer do obiektu na odpowiednim torze stacji
	"Cip".obiekt[#nr].nazwaObiektu := 'C2A1LH01';
	"Cip".obiekt[#nr].typObiektu := 9;
	"Cip".obiekt[#nr].inJestPotwWysterowania := 1;
	"Cip".obiekt[#nr].diPotwWysterowania := NOT "diC2A1LH01";
	#bool := "Cip".obiekt[#nr].hmiPotwWysterowania;
	// //
	 #nr := 105;//tu wpisz nuemr obiektu
	 "Cip".tor[0].zbiornikKwasu.czujnikDolnegoPoziomu := #nr; ;//tu przyporządkuj numer do obiektu na odpowiednim torze stacji
	 "Cip".obiekt[#nr].nazwaObiektu := 'C2A1LL01';
	 "Cip".obiekt[#nr].typObiektu := 9;
	 "Cip".obiekt[#nr].inJestPotwWysterowania := 1;
	 "Cip".obiekt[#nr].diPotwWysterowania :=  "diC2A1LL01";
	 #bool := "Cip".obiekt[#nr].hmiPotwWysterowania;
	//
	#nr := 43;//tu wpisz nuemr obiektu
	"Cip".tor[0].zbiorniczekDozowaniaKwasu.czujnikDolnegoPoziomu := #nr; ;//tu przyporządkuj numer do obiektu na odpowiednim torze stacji
	"Cip".obiekt[#nr].nazwaObiektu := 'C2A1LL41';
	"Cip".obiekt[#nr].typObiektu := 9;
	"Cip".obiekt[#nr].inJestPotwWysterowania := 1;
	"Cip".obiekt[#nr].diPotwWysterowania :=  "diC2A1LL41";
	#bool := "Cip".obiekt[#nr].hmiPotwWysterowania;
	// //
	// 
	
	
	#nr := 44;//tu wpisz nuemr obiektu
	"Cip".tor[0].zbiornikKwasu.czujnikwłazu := #nr; ;//tu przyporządkuj numer do obiektu na odpowiednim torze stacji
	"Cip".obiekt[#nr].nazwaObiektu := 'C2A1PD01';
	"Cip".obiekt[#nr].typObiektu := 9;
	"Cip".obiekt[#nr].inJestPotwWysterowania := 1;
	"Cip".obiekt[#nr].diPotwWysterowania := "diC2A1PD01";
	#bool := "Cip".obiekt[#nr].hmiPotwWysterowania;// //
	
	#nr := 50;//tu wpisz nuemr obiektu
	"Cip".tor[1].zbiornikDezynfekantu.czujnikGórnegoPoziomu := #nr; ;//tu przyporządkuj numer do obiektu na odpowiednim torze stacji
	"Cip".obiekt[#nr].nazwaObiektu := 'C2D1LH01';
	"Cip".obiekt[#nr].typObiektu := 9;
	"Cip".obiekt[#nr].inJestPotwWysterowania := 1;
	"Cip".obiekt[#nr].diPotwWysterowania :=NOT "diC2D1LH01";
	#bool := "Cip".obiekt[#nr].hmiPotwWysterowania;// //
	
	#nr := 51;//tu wpisz nuemr obiektu
	"Cip".tor[1].zbiornikDezynfekantu.czujnikDolnegoPoziomu  := #nr; ;//tu przyporządkuj numer do obiektu na odpowiednim torze stacji
	"Cip".obiekt[#nr].nazwaObiektu := 'C2D1LL01';
	"Cip".obiekt[#nr].typObiektu := 9;
	"Cip".obiekt[#nr].inJestPotwWysterowania := 1;
	"Cip".obiekt[#nr].diPotwWysterowania := "diC2D1LL01";
	#bool := "Cip".obiekt[#nr].hmiPotwWysterowania;// //
	
	#nr := 52;//tu wpisz nuemr obiektu
	"Cip".tor[1].zbiorniczekDozowanieDezynfekantu.czujnikDolnegoPoziomu:= #nr; ;//tu przyporządkuj numer do obiektu na odpowiednim torze stacji
	"Cip".obiekt[#nr].nazwaObiektu := 'C2D1LL81';
	"Cip".obiekt[#nr].typObiektu := 9;
	"Cip".obiekt[#nr].inJestPotwWysterowania := 1;
	"Cip".obiekt[#nr].diPotwWysterowania := "diC2D1LL81";
	#bool := "Cip".obiekt[#nr].hmiPotwWysterowania;// //
	
	#nr :=53;//tu wpisz nuemr obiektu
	"Cip".tor[1].zbiornikDezynfekantu.czujnikwłazu  := #nr; ;//tu przyporządkuj numer do obiektu na odpowiednim torze stacji
	"Cip".obiekt[#nr].nazwaObiektu := 'C2D1PD01';
	"Cip".obiekt[#nr].typObiektu := 9;
	"Cip".obiekt[#nr].inJestPotwWysterowania := 1;
	"Cip".obiekt[#nr].diPotwWysterowania := "diC2D1PD01";
	#bool := "Cip".obiekt[#nr].hmiPotwWysterowania;// //
	
	
	#nr := 59;//tu wpisz nuemr obiektu
	"Cip".tor[2].zbiornikDezynfekantu.czujnikGórnegoPoziomu := #nr; ;//tu przyporządkuj numer do obiektu na odpowiednim torze stacji
	"Cip".obiekt[#nr].nazwaObiektu := 'C2D2LH01';
	"Cip".obiekt[#nr].typObiektu := 9;
	"Cip".obiekt[#nr].inJestPotwWysterowania := 1;
	"Cip".obiekt[#nr].diPotwWysterowania :=NOT "diC2D2LH01";
	#bool := "Cip".obiekt[#nr].hmiPotwWysterowania;// //
	
	
	
	#nr := 60;//tu wpisz nuemr obiektu
	"Cip".tor[2].zbiornikDezynfekantu.czujnikDolnegoPoziomu := #nr; ;//tu przyporządkuj numer do obiektu na odpowiednim torze stacji
	"Cip".obiekt[#nr].nazwaObiektu := 'C2D2LL01';
	"Cip".obiekt[#nr].typObiektu := 9;
	"Cip".obiekt[#nr].inJestPotwWysterowania := 1;
	"Cip".obiekt[#nr].diPotwWysterowania := "diC2D2LL01";
	#bool := "Cip".obiekt[#nr].hmiPotwWysterowania;// //
	
	#nr := 61;//tu wpisz nuemr obiektu
	"Cip".tor[2].zbiorniczekDozowanieDezynfekantu.czujnikDolnegoPoziomu:= #nr; ;//tu przyporządkuj numer do obiektu na odpowiednim torze stacji
	"Cip".obiekt[#nr].nazwaObiektu := 'C2D2LL81';
	"Cip".obiekt[#nr].typObiektu := 9;
	"Cip".obiekt[#nr].inJestPotwWysterowania := 1;
	"Cip".obiekt[#nr].diPotwWysterowania := "diC2D2LL81";
	#bool := "Cip".obiekt[#nr].hmiPotwWysterowania;
	
	#nr := 62;//tu wpisz nuemr obiektu
	"Cip".tor[2].zbiornikDezynfekantu.czujnikwłazu:= #nr; ;//tu przyporządkuj numer do obiektu na odpowiednim torze stacji
	;//tu wpisz nazwę
	"Cip".obiekt[#nr].nazwaObiektu := 'C2D2PD01';
	"Cip".obiekt[#nr].typObiektu := 9;
	"Cip".obiekt[#nr].inJestPotwWysterowania := 1;
	"Cip".obiekt[#nr].diPotwWysterowania := "diC2D2PD01";
	#bool := "Cip".obiekt[#nr].hmiPotwWysterowania;// //
	
	
	#nr := 69;//tu wpisz nuemr obiektu
	"Cip".tor[1].zbiornikDezynfekantu_2.czujnikGórnegoPoziomu := #nr; ;//tu przyporządkuj numer do obiektu na odpowiednim torze stacji
	;//tu wpisz nazwę
	"Cip".obiekt[#nr].nazwaObiektu := 'C2D3LH01';
	"Cip".obiekt[#nr].typObiektu := 9;
	"Cip".obiekt[#nr].inJestPotwWysterowania := 1;
	"Cip".obiekt[#nr].diPotwWysterowania :=NOT "diC2D3LH01";
	#bool := "Cip".obiekt[#nr].hmiPotwWysterowania;// //
	
	#nr := 70;//tu wpisz nuemr obiektu
	"Cip".tor[1].zbiornikDezynfekantu_2.czujnikDolnegoPoziomu := #nr; ;//tu przyporządkuj numer do obiektu na odpowiednim torze stacji
	;//tu wpisz nazwę
	"Cip".obiekt[#nr].nazwaObiektu := 'C2D3LL01';
	"Cip".obiekt[#nr].typObiektu := 9;
	"Cip".obiekt[#nr].inJestPotwWysterowania := 1;
	"Cip".obiekt[#nr].diPotwWysterowania := "diC2L1LL01";
	#bool := "Cip".obiekt[#nr].hmiPotwWysterowania;// //
	
	#nr := 71;//tu wpisz nuemr obiektu
	"Cip".tor[1].zbiornikDezynfekantu_2.czujnikwłazu:= #nr; ;//tu przyporządkuj numer do obiektu na odpowiednim torze stacji
	;//tu wpisz nazwę
	"Cip".obiekt[#nr].nazwaObiektu := 'C2D3PD01';
	"Cip".obiekt[#nr].typObiektu := 9;
	"Cip".obiekt[#nr].inJestPotwWysterowania := 1;
	"Cip".obiekt[#nr].diPotwWysterowania := "diC2D3PD01";
	#bool := "Cip".obiekt[#nr].hmiPotwWysterowania;// //
	
	#nr := 79;//tu wpisz nuemr obiektu
	"Cip".tor[0].zbiornikŁugu.czujnikGórnegoPoziomu := #nr; ;//tu przyporządkuj numer do obiektu na odpowiednim torze stacji
	;//tu wpisz nazwę
	"Cip".obiekt[#nr].nazwaObiektu := 'C2L1LH01';
	"Cip".obiekt[#nr].typObiektu := 9;
	"Cip".obiekt[#nr].inJestPotwWysterowania := 1;
	"Cip".obiekt[#nr].diPotwWysterowania :=NOT "diC2L1LH01";
	#bool := "Cip".obiekt[#nr].hmiPotwWysterowania;// //
	
	#nr := 80;//tu wpisz nuemr obiektu
	"Cip".tor[0].zbiornikŁugu.czujnikDolnegoPoziomu := #nr; ;//tu przyporządkuj numer do obiektu na odpowiednim torze stacji
	;//tu wpisz nazwę
	"Cip".obiekt[#nr].nazwaObiektu := 'C2L1Ll01';
	"Cip".obiekt[#nr].typObiektu := 9;
	"Cip".obiekt[#nr].inJestPotwWysterowania := 1;
	"Cip".obiekt[#nr].diPotwWysterowania := "diC2D3LL01";
	#bool := "Cip".obiekt[#nr].hmiPotwWysterowania;// //
	
	#nr := 81;//tu wpisz nuemr obiektu
	"Cip".tor[0].zbiorniczekDozowaniaŁugu.czujnikDolnegoPoziomu := #nr; ;//tu przyporządkuj numer do obiektu na odpowiednim torze stacji
	;//tu wpisz nazwę
	"Cip".obiekt[#nr].nazwaObiektu := 'C2L1Ll41';
	"Cip".obiekt[#nr].typObiektu := 9;
	"Cip".obiekt[#nr].inJestPotwWysterowania := 1;
	"Cip".obiekt[#nr].diPotwWysterowania := "diC2L1LL41";
	#bool := "Cip".obiekt[#nr].hmiPotwWysterowania;// //
	
	#nr := 82;//tu wpisz nuemr obiektu
	"Cip".tor[0].zbiornikŁugu.czujnikwłazu := #nr; ;//tu przyporządkuj numer do obiektu na odpowiednim torze stacji
	;//tu wpisz nazwę
	"Cip".obiekt[#nr].nazwaObiektu := 'C2L1PD01';
	"Cip".obiekt[#nr].typObiektu := 9;
	"Cip".obiekt[#nr].inJestPotwWysterowania := 1;
	"Cip".obiekt[#nr].diPotwWysterowania := "diC2L1PD01";
	#bool := "Cip".obiekt[#nr].hmiPotwWysterowania;// //
	
	
	#nr := 88;//tu wpisz nuemr obiektu
	"Cip".tor[0].zbiornikWodyWtórnej.czujnikGórnegoPoziomu := #nr; ;//tu przyporządkuj numer do obiektu na odpowiednim torze stacji
	;//tu wpisz nazwę
	"Cip".obiekt[#nr].nazwaObiektu := 'C2R1LH01';
	"Cip".obiekt[#nr].typObiektu := 9;
	"Cip".obiekt[#nr].inJestPotwWysterowania := 1;
	"Cip".obiekt[#nr].diPotwWysterowania :=NOT "diC2R1LH01";
	#bool := "Cip".obiekt[#nr].hmiPotwWysterowania;// //
	
	
	#nr := 89;//tu wpisz nuemr obiektu
	"Cip".tor[0].zbiornikWodyWtórnej.czujnikDolnegoPoziomu  := #nr; ;//tu przyporządkuj numer do obiektu na odpowiednim torze stacji
	;//tu wpisz nazwę
	"Cip".obiekt[#nr].nazwaObiektu := 'C2R1LL01';
	"Cip".obiekt[#nr].typObiektu := 9;
	"Cip".obiekt[#nr].inJestPotwWysterowania := 1;
	"Cip".obiekt[#nr].diPotwWysterowania := "diC2R1LL01";
	#bool := "Cip".obiekt[#nr].hmiPotwWysterowania;// //
	
	#nr := 90;//tu wpisz nuemr obiektu
	"Cip".tor[0].zbiornikWodyWtórnej.czujnikwłazu  := #nr; ;//tu przyporządkuj numer do obiektu na odpowiednim torze stacji
	;//tu wpisz nazwę
	"Cip".obiekt[#nr].nazwaObiektu := 'C2R1PD01';
	"Cip".obiekt[#nr].typObiektu := 9;
	"Cip".obiekt[#nr].inJestPotwWysterowania := 1;
	"Cip".obiekt[#nr].diPotwWysterowania := "diC2R1PD01";
	#bool := "Cip".obiekt[#nr].hmiPotwWysterowania;// //
	
	#nr := 94;//tu wpisz nuemr obiektu
	"Cip".tor[0].zbiornikwodyCzystej.czujnikGórnegoPoziomu := #nr; ;//tu przyporządkuj numer do obiektu na odpowiednim torze stacji
	;//tu wpisz nazwę
	"Cip".obiekt[#nr].nazwaObiektu := 'C2W1LH01';
	"Cip".obiekt[#nr].typObiektu := 9;
	"Cip".obiekt[#nr].inJestPotwWysterowania := 1;
	"Cip".obiekt[#nr].diPotwWysterowania :=NOT "diC2W1LH01";
	#bool := "Cip".obiekt[#nr].hmiPotwWysterowania;// //
	
	
	#nr := 95;//tu wpisz nuemr obiektu
	"Cip".tor[0].zbiornikwodyCzystej.czujnikDolnegoPoziomu := #nr; ;//tu przyporządkuj numer do obiektu na odpowiednim torze stacji
	;//tu wpisz nazwę
	"Cip".obiekt[#nr].nazwaObiektu := 'C2W1LL01';
	"Cip".obiekt[#nr].typObiektu := 9;
	"Cip".obiekt[#nr].inJestPotwWysterowania := 1;
	"Cip".obiekt[#nr].diPotwWysterowania := "diC2W1LL01";
	#bool := "Cip".obiekt[#nr].hmiPotwWysterowania;// //
	
	#nr := 96;//tu wpisz nuemr obiektu
	"Cip".tor[0].zbiornikwodyCzystej.czujnikwłazu := #nr; ;//tu przyporządkuj numer do obiektu na odpowiednim torze stacji
	;//tu wpisz nazwę
	"Cip".obiekt[#nr].nazwaObiektu := 'C2W1PD01';
	"Cip".obiekt[#nr].typObiektu := 9;
	"Cip".obiekt[#nr].inJestPotwWysterowania := 1;
	"Cip".obiekt[#nr].diPotwWysterowania := "diC2W1PD01";
	#bool := "Cip".obiekt[#nr].hmiPotwWysterowania;// //
	
	
	#nr := 101;//tu wpisz nuemr obiektu
	"Cip".tor[1].czujnikPrzepływuNaPowrocie:= #nr; ;//tu przyporządkuj numer do obiektu na odpowiednim torze stacji
	;//tu wpisz nazwę
	"Cip".obiekt[#nr].nazwaObiektu := 'C211FV01';
	"Cip".obiekt[#nr].typObiektu := 9;
	"Cip".obiekt[#nr].inJestPotwWysterowania := 1;
	"Cip".obiekt[#nr].diPotwWysterowania := "diC211FV01";
	#bool := "Cip".obiekt[#nr].hmiPotwWysterowania;// //
	
	#nr := 102;//tu wpisz nuemr obiektu
	"Cip".tor[2].czujnikPrzepływuNaPowrocie:= #nr; ;//tu przyporządkuj numer do obiektu na odpowiednim torze stacji
	;//tu wpisz nazwę
	"Cip".obiekt[#nr].nazwaObiektu := 'C212FV01';
	"Cip".obiekt[#nr].typObiektu := 9;
	"Cip".obiekt[#nr].inJestPotwWysterowania := 1;
	"Cip".obiekt[#nr].diPotwWysterowania := "diC212FV01";
	#bool := "Cip".obiekt[#nr].hmiPotwWysterowania;// //
	
	
	#nr := 103;//tu wpisz nuemr obiektu
	"Cip".tor[1].czujnikPrzepływuDozowanegoDezynfekantu := #nr; ;//tu przyporządkuj numer do obiektu na odpowiednim torze stacji
	;//tu wpisz nazwę
	"Cip".obiekt[#nr].nazwaObiektu := 'C2D1FV81';
	"Cip".obiekt[#nr].typObiektu := 9;
	"Cip".obiekt[#nr].inJestPotwWysterowania := 1;
	"Cip".obiekt[#nr].diPotwWysterowania := "diC2D1FV81";
	#bool := "Cip".obiekt[#nr].hmiPotwWysterowania;// //
	
	#nr := 104;//tu wpisz nuemr obiektu
	"Cip".tor[2].czujnikPrzepływuDozowanegoDezynfekantu:= #nr; ;//tu przyporządkuj numer do obiektu na odpowiednim torze stacji
	;//tu wpisz nazwę
	"Cip".obiekt[#nr].nazwaObiektu := 'C2D2FV81';
	"Cip".obiekt[#nr].typObiektu := 9;
	"Cip".obiekt[#nr].inJestPotwWysterowania := 1;
	"Cip".obiekt[#nr].diPotwWysterowania := "diC2D2FV81";
	#bool := "Cip".obiekt[#nr].hmiPotwWysterowania;// //
	
	
	
	// // ///////////////////////zawory ONOFF i mix proof
	// // //
	// // //
	 #nr:=23 ;//tu wpisz nuemr obiektu
	 "Cip".tor[1].zawórBypassPrzygotowaniaStacji := #nr; ;//tu przyporządkuj numer do obiektu na odpowiednim torze stacji
	 "Cip".obiekt[#nr].nazwaObiektu := 'C201AV01';
	 "Cip".obiekt[#nr].typObiektu := 1;
	 "Cip".obiekt[#nr].inZezwolenieNaPracę := #diKSB_OK;
	 "Cip".obiekt[#nr].inJestPotwNiewysterowania := 0;
	 "Cip".obiekt[#nr].diPotwNieWysterowania :=0;
	 "Cip".obiekt[#nr].inJestPotwWysterowania := 1;
	 "Cip".obiekt[#nr].diPotwWysterowania := "diC201AV01c";
	 "doC201AV01b" := "Cip".obiekt[#nr].outStartUrządzenie;
	// // //
	#nr := 24;//tu wpisz nuemr obiektu
	"Cip".tor[1].zawórWydawczyCip := #nr; ;//tu przyporządkuj numer do obiektu na odpowiednim torze stacji
	;//tu wpisz nazwę
	"Cip".obiekt[#nr].nazwaObiektu := 'C201AV02';
	"Cip".obiekt[#nr].typObiektu := 1;
	"Cip".obiekt[#nr].inZezwolenieNaPracę := #diKSB_OK;
	"Cip".obiekt[#nr].inJestPotwNiewysterowania := 0;
	"Cip".obiekt[#nr].diPotwNieWysterowania := 0;
	"Cip".obiekt[#nr].inJestPotwWysterowania := 1;
	"Cip".obiekt[#nr].diPotwWysterowania := "diC201AV02c";
	"doC201AV02b" := "Cip".obiekt[#nr].outStartUrządzenie;
	// // //
	#nr := 25;//tu wpisz nuemr obiektu
	"Cip".tor[1].zawórParowyOdcinający:= #nr; ;//tu przyporządkuj numer do obiektu na odpowiednim torze stacji
	;//tu wpisz nazwę
	"Cip".obiekt[#nr].nazwaObiektu := 'C201AV21';
	"Cip".obiekt[#nr].typObiektu := 1;
	"Cip".obiekt[#nr].inZezwolenieNaPracę := #diKSB_OK;
	"Cip".obiekt[#nr].inJestPotwNiewysterowania := 0;
	"Cip".obiekt[#nr].diPotwNieWysterowania := 0;
	"Cip".obiekt[#nr].inJestPotwWysterowania := 0;
	"Cip".obiekt[#nr].diPotwWysterowania := 0;
	"doC201AV21b" := "Cip".obiekt[#nr].outStartUrządzenie;
	// // //
	#nr := 26;//tu wpisz nuemr obiektu
	"Cip".tor[2].zawórBypassPrzygotowaniaStacji := #nr; ;//tu przyporządkuj numer do obiektu na odpowiednim torze stacji
	;//tu wpisz nazwę
	"Cip".obiekt[#nr].nazwaObiektu := 'C202AV01';
	"Cip".obiekt[#nr].typObiektu := 1;
	"Cip".obiekt[#nr].inZezwolenieNaPracę := #diKSB_OK;
	"Cip".obiekt[#nr].inJestPotwNiewysterowania := 0;
	"Cip".obiekt[#nr].diPotwNieWysterowania := 0;
	"Cip".obiekt[#nr].inJestPotwWysterowania := 1;
	"Cip".obiekt[#nr].diPotwWysterowania := "diC202AV01c";
	"doC202AV01b" := "Cip".obiekt[#nr].outStartUrządzenie;
	// // //
	#nr := 27;//tu wpisz nuemr obiektu
	"Cip".tor[2].zawórWydawczyCip := #nr; ;//tu przyporządkuj numer do obiektu na odpowiednim torze stacji
	;//tu wpisz nazwę
	"Cip".obiekt[#nr].nazwaObiektu := 'C202AV02';
	"Cip".obiekt[#nr].typObiektu := 1;
	"Cip".obiekt[#nr].inZezwolenieNaPracę := #diKSB_OK;
	"Cip".obiekt[#nr].inJestPotwNiewysterowania := 0;
	"Cip".obiekt[#nr].diPotwNieWysterowania := 0;
	"Cip".obiekt[#nr].inJestPotwWysterowania := 1;
	"Cip".obiekt[#nr].diPotwWysterowania := "diC202AV02c";
	"doC202AV02b" := "Cip".obiekt[#nr].outStartUrządzenie;
	// // //
	#nr := 28;//tu wpisz nuemr obiektu
	"Cip".tor[0].pompkaDozowaniaŁuguwLinię := #nr; ;//tu przyporządkuj numer do obiektu na odpowiednim torze stacji
	;//tu wpisz nazwę
	"Cip".obiekt[#nr].nazwaObiektu := 'C202AV03';
	"Cip".obiekt[#nr].typObiektu := 1;
	"Cip".obiekt[#nr].inZezwolenieNaPracę := #diKSB_OK;
	"Cip".obiekt[#nr].inJestPotwNiewysterowania := 0;
	"Cip".obiekt[#nr].diPotwNieWysterowania := 0;
	"Cip".obiekt[#nr].inJestPotwWysterowania := 1;
	"Cip".obiekt[#nr].diPotwWysterowania := "diC202AV03c";
	"doC202AV03b" := "Cip".obiekt[#nr].outStartUrządzenie;
	// // //
	#nr := 29;//tu wpisz nuemr obiektu
	"Cip".tor[0].pompkaDozowaniaŁuguwLinię := #nr; ;//tu przyporządkuj numer do obiektu na odpowiednim torze stacji
	;//tu wpisz nazwę
	"Cip".obiekt[#nr].nazwaObiektu := 'C202AV04';
	"Cip".obiekt[#nr].typObiektu := 1;
	"Cip".obiekt[#nr].inZezwolenieNaPracę := #diKSB_OK;
	"Cip".obiekt[#nr].inJestPotwNiewysterowania := 0;
	"Cip".obiekt[#nr].diPotwNieWysterowania := 0;
	"Cip".obiekt[#nr].inJestPotwWysterowania := 1;
	"Cip".obiekt[#nr].diPotwWysterowania := "diC202AV04c";
	"doC202AV04b" := "Cip".obiekt[#nr].outStartUrządzenie;
	// // //
	#nr := 30;//tu wpisz nuemr obiektu
	"Cip".tor[2].zawórParowyOdcinający := #nr; ;//tu przyporządkuj numer do obiektu na odpowiednim torze stacji
	;//tu wpisz nazwę
	"Cip".obiekt[#nr].nazwaObiektu := 'C202AV21';
	"Cip".obiekt[#nr].typObiektu := 1;
	"Cip".obiekt[#nr].inZezwolenieNaPracę := #diKSB_OK;
	"Cip".obiekt[#nr].inJestPotwNiewysterowania := 0;
	"Cip".obiekt[#nr].diPotwNieWysterowania := 0;
	"Cip".obiekt[#nr].inJestPotwWysterowania := 0;
	"Cip".obiekt[#nr].diPotwWysterowania := 0;
	"doC202AV21b" := "Cip".obiekt[#nr].outStartUrządzenie;
	
	// // //
	#nr := 33;//tu wpisz nuemr obiektu
	"Cip".tor[1].zawórZrzutowyDoKanalizacji := #nr; ;//tu przyporządkuj numer do obiektu na odpowiednim torze stacji
	;//tu wpisz nazwę
	"Cip".obiekt[#nr].nazwaObiektu := 'C211AV01';
	"Cip".obiekt[#nr].typObiektu := 1;
	"Cip".obiekt[#nr].inZezwolenieNaPracę := #diKSB_OK;
	"Cip".obiekt[#nr].inJestPotwNiewysterowania := 0;
	"Cip".obiekt[#nr].diPotwNieWysterowania := 0;
	"Cip".obiekt[#nr].inJestPotwWysterowania := 1;
	"Cip".obiekt[#nr].diPotwWysterowania := "diC211AV01c";
	"doC211AV01b" := "Cip".obiekt[#nr].outStartUrządzenie;
	
	// // //
	#nr := 34;//tu wpisz nuemr obiektu
	"Cip".tor[2].zawórZrzutowyDoKanalizacji := #nr; ;//tu przyporządkuj numer do obiektu na odpowiednim torze stacji
	;//tu wpisz nazwę
	"Cip".obiekt[#nr].nazwaObiektu := 'C212AV01';
	"Cip".obiekt[#nr].typObiektu := 1;
	"Cip".obiekt[#nr].inZezwolenieNaPracę := #diKSB_OK;
	"Cip".obiekt[#nr].inJestPotwNiewysterowania := 0;
	"Cip".obiekt[#nr].diPotwNieWysterowania := 0;
	"Cip".obiekt[#nr].inJestPotwWysterowania := 1;
	"Cip".obiekt[#nr].diPotwWysterowania := "diC212AV01c";
	"doC212AV01b" := "Cip".obiekt[#nr].outStartUrządzenie;
	
	
	// // //
	#nr := 35;//tu wpisz nuemr obiektu
	"Cip".tor[1].zawórWydawczyKwasu := #nr; ;//tu przyporządkuj numer do obiektu na odpowiednim torze stacji
	;//tu wpisz nazwę
	"Cip".obiekt[#nr].nazwaObiektu := 'C2A1AV01';
	"Cip".obiekt[#nr].typObiektu := 1;
	"Cip".obiekt[#nr].inZezwolenieNaPracę := #diKSB_OK;
	"Cip".obiekt[#nr].inJestPotwNiewysterowania := 0;
	"Cip".obiekt[#nr].diPotwNieWysterowania := 0;
	"Cip".obiekt[#nr].inJestPotwWysterowania := 1;
	"Cip".obiekt[#nr].diPotwWysterowania := "diC2A1AV01c";
	"doC2A1AV01b" := "Cip".obiekt[#nr].outStartUrządzenie;
	// // //
	#nr := 36;//tu wpisz nuemr obiektu
	"Cip".tor[2].zawórWydawczyKwasu := #nr; ;//tu przyporządkuj numer do obiektu na odpowiednim torze stacji
	;//tu wpisz nazwę
	"Cip".obiekt[#nr].nazwaObiektu := 'C2A1AV02';
	"Cip".obiekt[#nr].typObiektu := 1;
	"Cip".obiekt[#nr].inZezwolenieNaPracę := #diKSB_OK;
	"Cip".obiekt[#nr].inJestPotwNiewysterowania := 0;
	"Cip".obiekt[#nr].diPotwNieWysterowania := 0;
	"Cip".obiekt[#nr].inJestPotwWysterowania := 1;
	"Cip".obiekt[#nr].diPotwWysterowania := "diC2A1AV02c";
	"doC2A1AV02b" := "Cip".obiekt[#nr].outStartUrządzenie;
	// // //
	#nr := 37;//tu wpisz nuemr obiektu
	"Cip".tor[1].zawórPowrotnyKwasu := #nr; ;//tu przyporządkuj numer do obiektu na odpowiednim torze stacji
	;//tu wpisz nazwę
	"Cip".obiekt[#nr].nazwaObiektu := 'C2A1AV11';
	"Cip".obiekt[#nr].typObiektu := 1;
	"Cip".obiekt[#nr].inZezwolenieNaPracę := #diKSB_OK;
	"Cip".obiekt[#nr].inJestPotwNiewysterowania := 0;
	"Cip".obiekt[#nr].diPotwNieWysterowania := 0;
	"Cip".obiekt[#nr].inJestPotwWysterowania := 1;
	"Cip".obiekt[#nr].diPotwWysterowania := "diC2A1AV11c";
	"doC2A1AV11b" := "Cip".obiekt[#nr].outStartUrządzenie;
	// // //
	#nr := 38;//tu wpisz nuemr obiektu
	"Cip".tor[2].zawórPowrotnyKwasu:= #nr; ;//tu przyporządkuj numer do obiektu na odpowiednim torze stacji
	;//tu wpisz nazwę
	"Cip".obiekt[#nr].nazwaObiektu := 'C2A1AV12';
	"Cip".obiekt[#nr].typObiektu := 1;
	"Cip".obiekt[#nr].inZezwolenieNaPracę := #diKSB_OK;
	"Cip".obiekt[#nr].inJestPotwNiewysterowania := 0;
	"Cip".obiekt[#nr].diPotwNieWysterowania := 0;
	"Cip".obiekt[#nr].inJestPotwWysterowania := 1;
	"Cip".obiekt[#nr].diPotwWysterowania := "diC2A1AV12c";
	"doC2A1AV12b" := "Cip".obiekt[#nr].outStartUrządzenie;
	// // //
	#nr := 39;//tu wpisz nuemr obiektu
	"Cip".tor[1].zawórUzupełnianiaWodyCzystejZbKwasu := #nr; ;//tu przyporządkuj numer do obiektu na odpowiednim torze stacji
	;//tu wpisz nazwę
	"Cip".obiekt[#nr].nazwaObiektu := 'C2A1AV31';
	"Cip".obiekt[#nr].typObiektu := 1;
	"Cip".obiekt[#nr].inZezwolenieNaPracę := #diKSB_OK;
	"Cip".obiekt[#nr].inJestPotwNiewysterowania := 0;
	"Cip".obiekt[#nr].diPotwNieWysterowania := 0;
	"Cip".obiekt[#nr].inJestPotwWysterowania := 1;
	"Cip".obiekt[#nr].diPotwWysterowania := "diC2A1AV31c";
	"doC2A1AV31b" := "Cip".obiekt[#nr].outStartUrządzenie;
	// // //
	#nr := 40;//tu wpisz nuemr obiektu
	"Cip".tor[1].zawórNaGruszkęZbiornikaKwasu := #nr; ;//tu przyporządkuj numer do obiektu na odpowiednim torze stacji
	;//tu wpisz nazwę
	"Cip".obiekt[#nr].nazwaObiektu := 'C2A1AV41';
	"Cip".obiekt[#nr].typObiektu := 1;
	"Cip".obiekt[#nr].inZezwolenieNaPracę := #diKSB_OK;
	"Cip".obiekt[#nr].inJestPotwNiewysterowania := 0;
	"Cip".obiekt[#nr].diPotwNieWysterowania := 0;
	"Cip".obiekt[#nr].inJestPotwWysterowania := 1;
	"Cip".obiekt[#nr].diPotwWysterowania := "diC2A1AV41c";
	"doC2A1AV41b" := "Cip".obiekt[#nr].outStartUrządzenie;
	// // //
	#nr := 41;//tu wpisz nuemr obiektu
	"Cip".tor[2].zawórDozowaniaKwasuwLinię:= #nr; ;//tu przyporządkuj numer do obiektu na odpowiednim torze stacji
	;//tu wpisz nazwę
	"Cip".obiekt[#nr].nazwaObiektu := 'C2A1AV42';
	"Cip".obiekt[#nr].typObiektu := 1;
	"Cip".obiekt[#nr].inZezwolenieNaPracę := #diKSB_OK;
	"Cip".obiekt[#nr].inJestPotwNiewysterowania := 0;
	"Cip".obiekt[#nr].diPotwNieWysterowania := 0;
	"Cip".obiekt[#nr].inJestPotwWysterowania := 0;
	"Cip".obiekt[#nr].diPotwWysterowania :=0;
	"doC2A1AV42b" := "Cip".obiekt[#nr].outStartUrządzenie;
	// // //
	#nr := 108;//tu wpisz nuemr obiektu
	"Cip".tor[1].pompkaDozowaniaKwasuwLinię := #nr; ;//tu przyporządkuj numer do obiektu na odpowiednim torze stacji
	;//tu wpisz nazwę
	"Cip".obiekt[#nr].nazwaObiektu := 'C2A1AV43';
	"Cip".obiekt[#nr].typObiektu := 1;
	"Cip".obiekt[#nr].inZezwolenieNaPracę := #diKSB_OK;
	"Cip".obiekt[#nr].inJestPotwNiewysterowania := 0;
	"Cip".obiekt[#nr].diPotwNieWysterowania := 0;
	"Cip".obiekt[#nr].inJestPotwWysterowania := 0;
	"Cip".obiekt[#nr].diPotwWysterowania := 0;
	"doC2A1AV43b" := "Cip".obiekt[#nr].outStartUrządzenie;
	// // //
	#nr := 109;//tu wpisz nuemr obiektu
	"Cip".tor[1].pompkaDozowaniaŁuguwLinię := #nr; ;//tu przyporządkuj numer do obiektu na odpowiednim torze stacji
	;//tu wpisz nazwę
	"Cip".obiekt[#nr].nazwaObiektu := 'C2L1AV43';
	"Cip".obiekt[#nr].typObiektu := 1;
	"Cip".obiekt[#nr].inZezwolenieNaPracę := #diKSB_OK;
	"Cip".obiekt[#nr].inJestPotwNiewysterowania := 0;
	"Cip".obiekt[#nr].diPotwNieWysterowania := 0;
	"Cip".obiekt[#nr].inJestPotwWysterowania := 0;
	"Cip".obiekt[#nr].diPotwWysterowania := 0;
	"doC2L1AV43b" := "Cip".obiekt[#nr].outStartUrządzenie;
	//
	#nr := 45;//tu wpisz nuemr obiektu
	"Cip".tor[1].zawórWydawczyDezynfekantu := #nr; ;//tu przyporządkuj numer do obiektu na odpowiednim torze stacji
	;//tu wpisz nazwę
	"Cip".obiekt[#nr].nazwaObiektu := 'C2D1AV01';
	"Cip".obiekt[#nr].typObiektu := 1;
	"Cip".obiekt[#nr].inZezwolenieNaPracę := #diKSB_OK;
	"Cip".obiekt[#nr].inJestPotwNiewysterowania := 0;
	"Cip".obiekt[#nr].diPotwNieWysterowania := 0;
	"Cip".obiekt[#nr].inJestPotwWysterowania := 1;
	"Cip".obiekt[#nr].diPotwWysterowania := "diC2D1AV01c";
	"doC2D1AV01b" := "Cip".obiekt[#nr].outStartUrządzenie;
	//
	#nr := 46;//tu wpisz nuemr obiektu
	"Cip".tor[1].zawórPowrotnyDezynfekantu := #nr; ;//tu przyporządkuj numer do obiektu na odpowiednim torze stacji
	;//tu wpisz nazwę
	"Cip".obiekt[#nr].nazwaObiektu := 'C2D1AV11';
	"Cip".obiekt[#nr].typObiektu := 1;
	"Cip".obiekt[#nr].inZezwolenieNaPracę := #diKSB_OK;
	"Cip".obiekt[#nr].inJestPotwNiewysterowania := 0;
	"Cip".obiekt[#nr].diPotwNieWysterowania := 0;
	"Cip".obiekt[#nr].inJestPotwWysterowania := 1;
	"Cip".obiekt[#nr].diPotwWysterowania := "diC2D1AV11c";
	"doC2D1AV11b" := "Cip".obiekt[#nr].outStartUrządzenie;
	//
	#nr := 47;//tu wpisz nuemr obiektu
	"Cip".tor[1].zawórStopowyPowrotuDezynfekantu := #nr; ;//tu przyporządkuj numer do obiektu na odpowiednim torze stacji
	;//tu wpisz nazwę
	"Cip".obiekt[#nr].nazwaObiektu := 'C2D1AV41';
	"Cip".obiekt[#nr].typObiektu := 1;
	"Cip".obiekt[#nr].inZezwolenieNaPracę := #diKSB_OK;
	"Cip".obiekt[#nr].inJestPotwNiewysterowania := 0;
	"Cip".obiekt[#nr].diPotwNieWysterowania := 0;
	"Cip".obiekt[#nr].inJestPotwWysterowania := 1;
	"Cip".obiekt[#nr].diPotwWysterowania := "diC2D1AV41c";
	"doC2D1AV41b" := "Cip".obiekt[#nr].outStartUrządzenie;
	//
	#nr := 48;//tu wpisz nuemr obiektu
	"Cip".tor[1].zawórNaGruszkęZbiornikaDezynfekantu := #nr; ;//tu przyporządkuj numer do obiektu na odpowiednim torze stacji
	;//tu wpisz nazwę
	"Cip".obiekt[#nr].nazwaObiektu := 'C2D1AV42';
	"Cip".obiekt[#nr].typObiektu := 1;
	"Cip".obiekt[#nr].inZezwolenieNaPracę := #diKSB_OK;
	"Cip".obiekt[#nr].inJestPotwNiewysterowania := 0;
	"Cip".obiekt[#nr].diPotwNieWysterowania := 0;
	"Cip".obiekt[#nr].inJestPotwWysterowania := 1;
	"Cip".obiekt[#nr].diPotwWysterowania := "diC2D1AV42c";
	"doC2D1AV42b" := "Cip".obiekt[#nr].outStartUrządzenie;
	//
	#nr := 49;//tu wpisz nuemr obiektu
	"Cip".tor[1].zawórDozowaniaDezynfekantuwLinię := #nr; ;//tu przyporządkuj numer do obiektu na odpowiednim torze stacji
	;//tu wpisz nazwę
	"Cip".obiekt[#nr].nazwaObiektu := 'C2D1AV81';
	"Cip".obiekt[#nr].typObiektu := 1;
	"Cip".obiekt[#nr].inZezwolenieNaPracę := #diKSB_OK;
	"Cip".obiekt[#nr].inJestPotwNiewysterowania := 0;
	"Cip".obiekt[#nr].diPotwNieWysterowania := 0;
	"Cip".obiekt[#nr].inJestPotwWysterowania := 0;
	"Cip".obiekt[#nr].diPotwWysterowania := 0;
	"doC2D1AV81b" := "Cip".obiekt[#nr].outStartUrządzenie;
	//
	#nr := 54;//tu wpisz nuemr obiektu
	"Cip".tor[2].zawórWydawczyDezynfekantu := #nr; ;//tu przyporządkuj numer do obiektu na odpowiednim torze stacji
	;//tu wpisz nazwę
	"Cip".obiekt[#nr].nazwaObiektu := 'C2D2AV01';
	"Cip".obiekt[#nr].typObiektu := 1;
	"Cip".obiekt[#nr].inZezwolenieNaPracę := #diKSB_OK;
	"Cip".obiekt[#nr].inJestPotwNiewysterowania := 0;
	"Cip".obiekt[#nr].diPotwNieWysterowania := 0;
	"Cip".obiekt[#nr].inJestPotwWysterowania := 1;
	"Cip".obiekt[#nr].diPotwWysterowania := "diC2D2AV01c";
	"doC2D2AV01b" := "Cip".obiekt[#nr].outStartUrządzenie;
	//
	#nr := 55;//tu wpisz nuemr obiektu
	"Cip".tor[2].zawórPowrotnyDezynfekantu := #nr; ;//tu przyporządkuj numer do obiektu na odpowiednim torze stacji
	;//tu wpisz nazwę
	"Cip".obiekt[#nr].nazwaObiektu := 'C2D2AV11';
	"Cip".obiekt[#nr].typObiektu := 1;
	"Cip".obiekt[#nr].inZezwolenieNaPracę := #diKSB_OK;
	"Cip".obiekt[#nr].inJestPotwNiewysterowania := 0;
	"Cip".obiekt[#nr].diPotwNieWysterowania := 0;
	"Cip".obiekt[#nr].inJestPotwWysterowania := 1;
	"Cip".obiekt[#nr].diPotwWysterowania := "diC2D2AV11c";
	"doC2D2AV11b" := "Cip".obiekt[#nr].outStartUrządzenie;
	//
	#nr := 56;//tu wpisz nuemr obiektu
	"Cip".tor[2].zawórStopowyPowrotuDezynfekantu := #nr; ;//tu przyporządkuj numer do obiektu na odpowiednim torze stacji
	;//tu wpisz nazwę
	"Cip".obiekt[#nr].nazwaObiektu := 'C2D2AV41';
	"Cip".obiekt[#nr].typObiektu := 1;
	"Cip".obiekt[#nr].inZezwolenieNaPracę := #diKSB_OK;
	"Cip".obiekt[#nr].inJestPotwNiewysterowania := 0;
	"Cip".obiekt[#nr].diPotwNieWysterowania := 0;
	"Cip".obiekt[#nr].inJestPotwWysterowania := 1;
	"Cip".obiekt[#nr].diPotwWysterowania := "diC2D2AV41c";
	"doC2D2AV41b" := "Cip".obiekt[#nr].outStartUrządzenie;
	//
	#nr := 57;//tu wpisz nuemr obiektu
	"Cip".tor[2].zawórNaGruszkęZbiornikaDezynfekantu := #nr; ;//tu przyporządkuj numer do obiektu na odpowiednim torze stacji
	;//tu wpisz nazwę
	"Cip".obiekt[#nr].nazwaObiektu := 'C2D2AV42';
	"Cip".obiekt[#nr].typObiektu := 1;
	"Cip".obiekt[#nr].inZezwolenieNaPracę := #diKSB_OK;
	"Cip".obiekt[#nr].inJestPotwNiewysterowania := 0;
	"Cip".obiekt[#nr].diPotwNieWysterowania := 0;
	"Cip".obiekt[#nr].inJestPotwWysterowania := 1;
	"Cip".obiekt[#nr].diPotwWysterowania := "diC2D2AV42c";
	"doC2D2AV42b" := "Cip".obiekt[#nr].outStartUrządzenie;
	//
	#nr := 58;//tu wpisz nuemr obiektu
	"Cip".tor[2].zawórDozowaniaDezynfekantuwLinię := #nr; ;//tu przyporządkuj numer do obiektu na odpowiednim torze stacji
	;//tu wpisz nazwę
	"Cip".obiekt[#nr].nazwaObiektu := 'C2D2AV81';
	"Cip".obiekt[#nr].typObiektu := 1;
	"Cip".obiekt[#nr].inZezwolenieNaPracę := #diKSB_OK;
	"Cip".obiekt[#nr].inJestPotwNiewysterowania := 0;
	"Cip".obiekt[#nr].diPotwNieWysterowania := 0;
	"Cip".obiekt[#nr].inJestPotwWysterowania :=0;
	"Cip".obiekt[#nr].diPotwWysterowania := 0;
	"doC2D2AV81b" := "Cip".obiekt[#nr].outStartUrządzenie;
	//
	#nr := 63;//tu wpisz nuemr obiektu
	"Cip".tor[1].zawórWydawczyDezynfekantu_2 := #nr; ;//tu przyporządkuj numer do obiektu na odpowiednim torze stacji
	;//tu wpisz nazwę
	"Cip".obiekt[#nr].nazwaObiektu := 'C2D3AV01';
	"Cip".obiekt[#nr].typObiektu := 1;
	"Cip".obiekt[#nr].inZezwolenieNaPracę := #diKSB_OK;
	"Cip".obiekt[#nr].inJestPotwNiewysterowania := 0;
	"Cip".obiekt[#nr].diPotwNieWysterowania := 0;
	"Cip".obiekt[#nr].inJestPotwWysterowania := 1;
	"Cip".obiekt[#nr].diPotwWysterowania := "diC2D3AV01c";
	"doC2D3AV01b" := "Cip".obiekt[#nr].outStartUrządzenie;
	//
	#nr := 64;//tu wpisz nuemr obiektu
	"Cip".tor[1].zawórStopowyPowrotuDezynfekantu_2:= #nr; ;//tu przyporządkuj numer do obiektu na odpowiednim torze stacji
	;//tu wpisz nazwę
	"Cip".obiekt[#nr].nazwaObiektu := 'C2D3AV11';
	"Cip".obiekt[#nr].typObiektu := 1;
	"Cip".obiekt[#nr].inZezwolenieNaPracę := #diKSB_OK;
	"Cip".obiekt[#nr].inJestPotwNiewysterowania := 0;
	"Cip".obiekt[#nr].diPotwNieWysterowania := 0;
	"Cip".obiekt[#nr].inJestPotwWysterowania := 1;
	"Cip".obiekt[#nr].diPotwWysterowania := "diC2D3AV11c";
	"doC2D3AV11b" := "Cip".obiekt[#nr].outStartUrządzenie;
	//
	#nr := 65;//tu wpisz nuemr obiektu
	"Cip".tor[1].ZawórUzupełnianiaWodyCzystejZbDezynfekantu_2 := #nr;//tu przyporządkuj numer do obiektu na odpowiednim torze stacji
	"Cip".obiekt[#nr].nazwaObiektu := 'C2D3AV31';
	"Cip".obiekt[#nr].typObiektu := 1;
	"Cip".obiekt[#nr].inZezwolenieNaPracę := #diKSB_OK;
	"Cip".obiekt[#nr].inJestPotwNiewysterowania := 0;
	"Cip".obiekt[#nr].diPotwNieWysterowania := 0;
	"Cip".obiekt[#nr].inJestPotwWysterowania := 1;
	"Cip".obiekt[#nr].diPotwWysterowania := "diC2D3AV31c";
	"doC2D3AV31b" := "Cip".obiekt[#nr].outStartUrządzenie;
	//
	#nr := 66;//tu wpisz nuemr obiektu
	"Cip".tor[1].zawórStopowyPowrotuDezynfekantu_2 := #nr; ;//tu przyporządkuj numer do obiektu na odpowiednim torze stacji
	;//tu wpisz nazwę
	"Cip".obiekt[#nr].nazwaObiektu := 'C2D3AV41';
	"Cip".obiekt[#nr].typObiektu := 1;
	"Cip".obiekt[#nr].inZezwolenieNaPracę := #diKSB_OK;
	"Cip".obiekt[#nr].inJestPotwNiewysterowania := 0;
	"Cip".obiekt[#nr].diPotwNieWysterowania := 0;
	"Cip".obiekt[#nr].inJestPotwWysterowania := 1;
	"Cip".obiekt[#nr].diPotwWysterowania := "diC2D3AV41c";
	"doC2D3AV41b" := "Cip".obiekt[#nr].outStartUrządzenie;
	//
	#nr := 67;//tu wpisz nuemr obiektu
	"Cip".tor[1].zawórNaGruszkęZbiornikaDezynfekantu_2 := #nr; ;//tu przyporządkuj numer do obiektu na odpowiednim torze stacji
	;//tu wpisz nazwę
	"Cip".obiekt[#nr].nazwaObiektu := 'C2D3AV42';
	"Cip".obiekt[#nr].typObiektu := 1;
	"Cip".obiekt[#nr].inZezwolenieNaPracę := #diKSB_OK;
	"Cip".obiekt[#nr].inJestPotwNiewysterowania := 0;
	"Cip".obiekt[#nr].diPotwNieWysterowania := 0;
	"Cip".obiekt[#nr].inJestPotwWysterowania := 1;
	"Cip".obiekt[#nr].diPotwWysterowania := "diC2D3AV42c";
	"doC2D3AV42b" := "Cip".obiekt[#nr].outStartUrządzenie;
	//
	#nr := 68;//tu wpisz nuemr obiektu
	"Cip".tor[1].zawórWodaNaGruszkęZbiornikaDezynfekantu_2 := #nr; ;//tu przyporządkuj numer do obiektu na odpowiednim torze stacji
	;//tu wpisz nazwę
	"Cip".obiekt[#nr].nazwaObiektu := 'C2D3AV43';
	"Cip".obiekt[#nr].typObiektu := 1;
	"Cip".obiekt[#nr].inZezwolenieNaPracę := #diKSB_OK;
	"Cip".obiekt[#nr].inJestPotwNiewysterowania := 0;
	"Cip".obiekt[#nr].diPotwNieWysterowania := 0;
	"Cip".obiekt[#nr].inJestPotwWysterowania := 1;
	"Cip".obiekt[#nr].diPotwWysterowania := "diC2D3AV43c";
	"doC2D3AV43b" := "Cip".obiekt[#nr].outStartUrządzenie;
	//
	#nr :=72;//tu wpisz nuemr obiektu
	"Cip".tor[1].zawórWydawczyŁugu := #nr; ;//tu przyporządkuj numer do obiektu na odpowiednim torze stacji
	;//tu wpisz nazwę
	"Cip".obiekt[#nr].nazwaObiektu := 'C2L1AV01';
	"Cip".obiekt[#nr].typObiektu := 1;
	"Cip".obiekt[#nr].inZezwolenieNaPracę := #diKSB_OK;
	"Cip".obiekt[#nr].inJestPotwNiewysterowania := 0;
	"Cip".obiekt[#nr].diPotwNieWysterowania := 0;
	"Cip".obiekt[#nr].inJestPotwWysterowania := 1;
	"Cip".obiekt[#nr].diPotwWysterowania := "diC2L1AV01c";
	"doC2L1AV01b" := "Cip".obiekt[#nr].outStartUrządzenie;
	//
	#nr := 73;//tu wpisz nuemr obiektu
	"Cip".tor[2].zawórWydawczyŁugu := #nr; ;//tu przyporządkuj numer do obiektu na odpowiednim torze stacji
	;//tu wpisz nazwę
	"Cip".obiekt[#nr].nazwaObiektu := 'C2L1AV02';
	"Cip".obiekt[#nr].typObiektu := 1;
	"Cip".obiekt[#nr].inZezwolenieNaPracę := #diKSB_OK;
	"Cip".obiekt[#nr].inJestPotwNiewysterowania := 0;
	"Cip".obiekt[#nr].diPotwNieWysterowania := 0;
	"Cip".obiekt[#nr].inJestPotwWysterowania := 1;
	"Cip".obiekt[#nr].diPotwWysterowania := "diC2L1AV02c";
	"doC2L1AV02b" := "Cip".obiekt[#nr].outStartUrządzenie;
	//
	#nr := 74;//tu wpisz nuemr obiektu
	"Cip".tor[1].zawórPowrotnyŁugu := #nr; ;//tu przyporządkuj numer do obiektu na odpowiednim torze stacji
	;//tu wpisz nazwę
	"Cip".obiekt[#nr].nazwaObiektu := 'C2L1AV11';
	"Cip".obiekt[#nr].typObiektu := 1;
	"Cip".obiekt[#nr].inZezwolenieNaPracę := #diKSB_OK;
	"Cip".obiekt[#nr].inJestPotwNiewysterowania := 0;
	"Cip".obiekt[#nr].diPotwNieWysterowania := 0;
	"Cip".obiekt[#nr].inJestPotwWysterowania := 1;
	"Cip".obiekt[#nr].diPotwWysterowania := "diC2L1AV11c";
	"doC2L1AV11b" := "Cip".obiekt[#nr].outStartUrządzenie;
	//
	#nr := 75;//tu wpisz nuemr obiektu
	"Cip".tor[2].zawórPowrotnyŁugu := #nr; ;//tu przyporządkuj numer do obiektu na odpowiednim torze stacji
	;//tu wpisz nazwę
	"Cip".obiekt[#nr].nazwaObiektu := 'C2L1AV12';
	"Cip".obiekt[#nr].typObiektu := 1;
	"Cip".obiekt[#nr].inZezwolenieNaPracę := #diKSB_OK;
	"Cip".obiekt[#nr].inJestPotwNiewysterowania := 0;
	"Cip".obiekt[#nr].diPotwNieWysterowania := 0;
	"Cip".obiekt[#nr].inJestPotwWysterowania := 1;
	"Cip".obiekt[#nr].diPotwWysterowania := "diC2L1AV12c";
	"doC2L1AV12b" := "Cip".obiekt[#nr].outStartUrządzenie;
	//
	#nr := 76;//tu wpisz nuemr obiektu
	"Cip".tor[1].zawórUzupełnianiaWodyCzystejZbŁugu := #nr; ;//tu przyporządkuj numer do obiektu na odpowiednim torze stacji
	;//tu wpisz nazwę
	"Cip".obiekt[#nr].nazwaObiektu := 'C2L1AV31';
	"Cip".obiekt[#nr].typObiektu := 1;
	"Cip".obiekt[#nr].inZezwolenieNaPracę := #diKSB_OK;
	"Cip".obiekt[#nr].inJestPotwNiewysterowania := 0;
	"Cip".obiekt[#nr].diPotwNieWysterowania := 0;
	"Cip".obiekt[#nr].inJestPotwWysterowania := 1;
	"Cip".obiekt[#nr].diPotwWysterowania := "diC2L1AV31c";
	"doC2L1AV31b" := "Cip".obiekt[#nr].outStartUrządzenie;
	//
	#nr := 77;//tu wpisz nuemr obiektu
	"Cip".tor[1].zawórNaGruszkęZbiornikaŁugu := #nr; ;//tu przyporządkuj numer do obiektu na odpowiednim torze stacji
	;//tu wpisz nazwę
	"Cip".obiekt[#nr].nazwaObiektu := 'C2L1AV41';
	"Cip".obiekt[#nr].typObiektu := 1;
	"Cip".obiekt[#nr].inZezwolenieNaPracę := #diKSB_OK;
	"Cip".obiekt[#nr].inJestPotwNiewysterowania := 0;
	"Cip".obiekt[#nr].diPotwNieWysterowania := 0;
	"Cip".obiekt[#nr].inJestPotwWysterowania := 1;
	"Cip".obiekt[#nr].diPotwWysterowania := "diC2L1AV41c";
	"doC2L1AV41b" := "Cip".obiekt[#nr].outStartUrządzenie;
	//
	#nr := 78;//tu wpisz nuemr obiektu
	"Cip".tor[2].zawórDozowaniaLuguwLinię := #nr; ;//tu przyporządkuj numer do obiektu na odpowiednim torze stacji
	;//tu wpisz nazwę
	"Cip".obiekt[#nr].nazwaObiektu := 'C2L1AV42';
	"Cip".obiekt[#nr].typObiektu := 1;
	"Cip".obiekt[#nr].inZezwolenieNaPracę := #diKSB_OK;
	"Cip".obiekt[#nr].inJestPotwNiewysterowania := 0;
	"Cip".obiekt[#nr].diPotwNieWysterowania := 0;
	"Cip".obiekt[#nr].inJestPotwWysterowania := 0;
	"Cip".obiekt[#nr].diPotwWysterowania :=1;
	"doC2L1AV42b" := "Cip".obiekt[#nr].outStartUrządzenie;
	//
	#nr := 83;//tu wpisz nuemr obiektu
	"Cip".tor[1].zawórWydawczyWodyWtórnej:= #nr; ;//tu przyporządkuj numer do obiektu na odpowiednim torze stacji
	;//tu wpisz nazwę
	"Cip".obiekt[#nr].nazwaObiektu := 'C2R1AV01';
	"Cip".obiekt[#nr].typObiektu := 1;
	"Cip".obiekt[#nr].inZezwolenieNaPracę := #diKSB_OK;
	"Cip".obiekt[#nr].inJestPotwNiewysterowania := 0;
	"Cip".obiekt[#nr].diPotwNieWysterowania := 0;
	"Cip".obiekt[#nr].inJestPotwWysterowania := 1;
	"Cip".obiekt[#nr].diPotwWysterowania := "diC2R1AV01c";
	"doC2R1AV01b" := "Cip".obiekt[#nr].outStartUrządzenie;
	//
	#nr := 84;//tu wpisz nuemr obiektu
	"Cip".tor[2].zawórWydawczyWodyWtórnej := #nr; ;//tu przyporządkuj numer do obiektu na odpowiednim torze stacji
	;//tu wpisz nazwę
	"Cip".obiekt[#nr].nazwaObiektu := 'C2R1AV02';
	"Cip".obiekt[#nr].typObiektu := 1;
	"Cip".obiekt[#nr].inZezwolenieNaPracę := #diKSB_OK;
	"Cip".obiekt[#nr].inJestPotwNiewysterowania := 0;
	"Cip".obiekt[#nr].diPotwNieWysterowania := 0;
	"Cip".obiekt[#nr].inJestPotwWysterowania := 1;
	"Cip".obiekt[#nr].diPotwWysterowania := "diC2R1AV02c";
	"doC2R1AV02b" := "Cip".obiekt[#nr].outStartUrządzenie;
	//
	#nr := 85;//tu wpisz nuemr obiektu
	"Cip".tor[1].zawórPowrotnyWodyWtórnej := #nr; ;//tu przyporządkuj numer do obiektu na odpowiednim torze stacji
	;//tu wpisz nazwę
	"Cip".obiekt[#nr].nazwaObiektu := 'C2R1AV11';
	"Cip".obiekt[#nr].typObiektu := 1;
	"Cip".obiekt[#nr].inZezwolenieNaPracę := #diKSB_OK;
	"Cip".obiekt[#nr].inJestPotwNiewysterowania := 0;
	"Cip".obiekt[#nr].diPotwNieWysterowania := 0;
	"Cip".obiekt[#nr].inJestPotwWysterowania := 1;
	"Cip".obiekt[#nr].diPotwWysterowania := "diC2R1AV11c";
	"doC2R1AV11b" := "Cip".obiekt[#nr].outStartUrządzenie;
	//
	#nr := 86;//tu wpisz nuemr obiektu
	"Cip".tor[2].zawórPowrotnyWodyWtórnej := #nr; ;//tu przyporządkuj numer do obiektu na odpowiednim torze stacji
	;//tu wpisz nazwę
	"Cip".obiekt[#nr].nazwaObiektu := 'C2R1AV12';
	"Cip".obiekt[#nr].typObiektu := 1;
	"Cip".obiekt[#nr].inZezwolenieNaPracę := #diKSB_OK;
	"Cip".obiekt[#nr].inJestPotwNiewysterowania := 0;
	"Cip".obiekt[#nr].diPotwNieWysterowania := 0;
	"Cip".obiekt[#nr].inJestPotwWysterowania := 1;
	"Cip".obiekt[#nr].diPotwWysterowania := "diC2R1AV12c";
	"doC2R1AV12b" := "Cip".obiekt[#nr].outStartUrządzenie;
	//
	#nr := 87;//tu wpisz nuemr obiektu
	"Cip".tor[1].zawórNaGruszkęZbiornikaWodyWtórnej := #nr; ;//tu przyporządkuj numer do obiektu na odpowiednim torze stacji
	;//tu wpisz nazwę
	"Cip".obiekt[#nr].nazwaObiektu := 'C2R1AV41';
	"Cip".obiekt[#nr].typObiektu := 1;
	"Cip".obiekt[#nr].inZezwolenieNaPracę := #diKSB_OK;
	"Cip".obiekt[#nr].inJestPotwNiewysterowania := 0;
	"Cip".obiekt[#nr].diPotwNieWysterowania := 0;
	"Cip".obiekt[#nr].inJestPotwWysterowania := 1;
	"Cip".obiekt[#nr].diPotwWysterowania := "diC2R1AV41c";
	"doC2R1AV41b" := "Cip".obiekt[#nr].outStartUrządzenie;
	//
	#nr := 91;//tu wpisz nuemr obiektu
	"Cip".tor[2].zawórWydawczyWodyCzystej := #nr; ;//tu przyporządkuj numer do obiektu na odpowiednim torze stacji
	;//tu wpisz nazwę
	"Cip".obiekt[#nr].nazwaObiektu := 'C2W1AV02';
	"Cip".obiekt[#nr].typObiektu := 1;
	"Cip".obiekt[#nr].inZezwolenieNaPracę := #diKSB_OK;
	"Cip".obiekt[#nr].inJestPotwNiewysterowania := 0;
	"Cip".obiekt[#nr].diPotwNieWysterowania := 0;
	"Cip".obiekt[#nr].inJestPotwWysterowania := 1;
	"Cip".obiekt[#nr].diPotwWysterowania := "diC2W1AV02c";
	"doC2W1AV02b" := "Cip".obiekt[#nr].outStartUrządzenie;
	//
	#nr := 92;//tu wpisz nuemr obiektu
	"Cip".tor[1].zawórUzupełnianiaWodyCzystejZbWodyCzystej := #nr; ;//tu przyporządkuj numer do obiektu na odpowiednim torze stacji
	;//tu wpisz nazwę
	"Cip".obiekt[#nr].nazwaObiektu := 'C2W1AV31';
	"Cip".obiekt[#nr].typObiektu := 1;
	"Cip".obiekt[#nr].inZezwolenieNaPracę := #diKSB_OK;
	"Cip".obiekt[#nr].inJestPotwNiewysterowania := 0;
	"Cip".obiekt[#nr].diPotwNieWysterowania := 0;
	"Cip".obiekt[#nr].inJestPotwWysterowania := 1;
	"Cip".obiekt[#nr].diPotwWysterowania := "diC2W1AV31c";
	"doC2W1AV31b" := "Cip".obiekt[#nr].outStartUrządzenie;
	//
	#nr := 93;//tu wpisz nuemr obiektu
	"Cip".tor[1].zawórNaGruszkęZbiornikaWodyCzystej := #nr; ;//tu przyporządkuj numer do obiektu na odpowiednim torze stacji
	;//tu wpisz nazwę
	"Cip".obiekt[#nr].nazwaObiektu := 'C2W1AV41';
	"Cip".obiekt[#nr].typObiektu := 1;
	"Cip".obiekt[#nr].inZezwolenieNaPracę := #diKSB_OK;
	"Cip".obiekt[#nr].inJestPotwNiewysterowania := 0;
	"Cip".obiekt[#nr].diPotwNieWysterowania := 0;
	"Cip".obiekt[#nr].inJestPotwWysterowania := 1;
	"Cip".obiekt[#nr].diPotwWysterowania := "diC2W1AV41c";
	"doC2W1AV41b" := "Cip".obiekt[#nr].outStartUrządzenie;
	//
	//
	#nr :=110;//tu wpisz nuemr obiektu
	"Cip".tor[1].zawórWydawczyWodyCzystej:= #nr; ;//tu przyporządkuj numer do obiektu na odpowiednim torze stacji
	;//tu wpisz nazwę
	"Cip".obiekt[#nr].nazwaObiektu := 'C2W1AV01';
	"Cip".obiekt[#nr].typObiektu := 1;
	"Cip".obiekt[#nr].inZezwolenieNaPracę := #diKSB_OK;
	"Cip".obiekt[#nr].inJestPotwNiewysterowania := 0;
	"Cip".obiekt[#nr].diPotwNieWysterowania := 0;
	"Cip".obiekt[#nr].inJestPotwWysterowania := 1;
	"Cip".obiekt[#nr].diPotwWysterowania := "diC2W1AV01c";
	"doC2W1AV01b" := "Cip".obiekt[#nr].outStartUrządzenie;
	
	
	
	
	// ////////////////////////temperatura
	//
	#nr:=1 ;//tu wpisz nuemr obiektu
	"Cip".tor[0].zbiornikwodyCzystej.temperatura := #nr; ;//tu przyporządkuj numer do obiektu na odpowiednim torze stacji
	"Cip".obiekt[#nr].nazwaObiektu := 'C2W1TT01';
	"Cip".obiekt[#nr].typObiektu := 5;
	"Cip".obiekt[#nr].inPomiarRaw := "aiC2W1TT01";
	#real := "Cip".obiekt[#nr].WartośćPomiaru;
	//
	#nr := 2;//tu wpisz nuemr obiektu
	"Cip".tor[0].zbiornikWodyWtórnej.temperatura := #nr; ;//tu przyporządkuj numer do obiektu na odpowiednim torze stacji
	;//tu wpisz nazwę
	"Cip".obiekt[#nr].nazwaObiektu := 'C2R1TT01';
	"Cip".obiekt[#nr].typObiektu := 5;
	"Cip".obiekt[#nr].inPomiarRaw := "aiC2R1TT01";
	#real := "Cip".obiekt[#nr].WartośćPomiaru;
	//
	#nr := 3;//tu wpisz nuemr obiektu
	"Cip".tor[0].zbiornikŁugu.temperatura := #nr; ;//tu przyporządkuj numer do obiektu na odpowiednim torze stacji
	;//tu wpisz nazwę
	"Cip".obiekt[#nr].nazwaObiektu := 'C2L1TT01';
	"Cip".obiekt[#nr].typObiektu := 5;
	"Cip".obiekt[#nr].inPomiarRaw := "aiC2L1TT01";
	#real := "Cip".obiekt[#nr].WartośćPomiaru;
	//
	#nr := 4;//tu wpisz nuemr obiektu
	"Cip".tor[0].zbiornikKwasu.temperatura := #nr; ;//tu przyporządkuj numer do obiektu na odpowiednim torze stacji
	;//tu wpisz nazwę
	"Cip".obiekt[#nr].nazwaObiektu := 'C2A1TT01';
	"Cip".obiekt[#nr].typObiektu := 5;
	"Cip".obiekt[#nr].inPomiarRaw := "aiC2A1TT01";
	#real := "Cip".obiekt[#nr].WartośćPomiaru;
	//
	#nr := 5;//tu wpisz nuemr obiektu
	"Cip".tor[1].zbiornikDezynfekantu.temperatura := #nr; ;//tu przyporządkuj numer do obiektu na odpowiednim torze stacji
	;//tu wpisz nazwę
	"Cip".obiekt[#nr].nazwaObiektu := 'C2D1TT01';
	"Cip".obiekt[#nr].typObiektu := 5;
	"Cip".obiekt[#nr].inPomiarRaw := "aiC2D1TT01";
	#real := "Cip".obiekt[#nr].WartośćPomiaru;
	//
	#nr := 6;//tu wpisz nuemr obiektu
	"Cip".tor[2].zbiornikDezynfekantu.temperatura:= #nr; ;//tu przyporządkuj numer do obiektu na odpowiednim torze stacji
	;//tu wpisz nazwę
	"Cip".obiekt[#nr].nazwaObiektu := 'C2D2TT01';
	"Cip".obiekt[#nr].typObiektu := 5;
	"Cip".obiekt[#nr].inPomiarRaw := "aiC2D2TT01";
	#real := "Cip".obiekt[#nr].WartośćPomiaru;
	//
	#nr := 7;//tu wpisz nuemr obiektu
	"Cip".tor[1].zbiornikDezynfekantu_2.temperatura := #nr; ;//tu przyporządkuj numer do obiektu na odpowiednim torze stacji
	;//tu wpisz nazwę
	"Cip".obiekt[#nr].nazwaObiektu := 'C2D3TT01';
	"Cip".obiekt[#nr].typObiektu := 5;
	"Cip".obiekt[#nr].inPomiarRaw := "aiC2D3TT01";
	#real := "Cip".obiekt[#nr].WartośćPomiaru;
	//
	#nr := 8;//tu wpisz nuemr obiektu
	"Cip".tor[1].temperaturaNaPowrocie:= #nr; ;//tu przyporządkuj numer do obiektu na odpowiednim torze stacji
	;//tu wpisz nazwę
	"Cip".obiekt[#nr].nazwaObiektu := 'C211TT01';
	"Cip".obiekt[#nr].typObiektu := 5;
	"Cip".obiekt[#nr].inPomiarRaw := "aiC211TT01";
	#real := "Cip".obiekt[#nr].WartośćPomiaru;
	//
	#nr := 9;//tu wpisz nuemr obiektu
	"Cip".tor[2].temperaturaNaPowrocie := #nr; ;//tu przyporządkuj numer do obiektu na odpowiednim torze stacji
	;//tu wpisz nazwę
	"Cip".obiekt[#nr].nazwaObiektu := 'C212TT01';
	"Cip".obiekt[#nr].typObiektu := 5;
	"Cip".obiekt[#nr].inPomiarRaw := "aiC212TT01";
	#real := "Cip".obiekt[#nr].WartośćPomiaru;
	//
	#nr := 10;//tu wpisz nuemr obiektu
	"Cip".tor[1].temperaturaZaWymiennikiem := #nr; ;//tu przyporządkuj numer do obiektu na odpowiednim torze stacji
	;//tu wpisz nazwę
	"Cip".obiekt[#nr].nazwaObiektu := 'C201TT01';
	"Cip".obiekt[#nr].typObiektu := 5;
	"Cip".obiekt[#nr].inPomiarRaw := "aiC201TT01";
	#real := "Cip".obiekt[#nr].WartośćPomiaru;
	//
	#nr := 11;//tu wpisz nuemr obiektu
	"Cip".tor[2].temperaturaZaWymiennikiem := #nr; ;//tu przyporządkuj numer do obiektu na odpowiednim torze stacji
	;//tu wpisz nazwę
	"Cip".obiekt[#nr].nazwaObiektu := 'C202TT01';
	"Cip".obiekt[#nr].typObiektu := 5;
	"Cip".obiekt[#nr].inPomiarRaw := "aiC202TT01";
	#real := "Cip".obiekt[#nr].WartośćPomiaru;
	
	// // //////////////////////mierniki poziomu
	// // //
	#nr:=14;//tu wpisz nuemr obiektu
	"Cip".tor[0].zbiornikKwasu.poziomAnalogowy := #nr; ;//tu przyporządkuj numer do obiektu na odpowiednim torze stacji
	"Cip".obiekt[#nr].nazwaObiektu := 'C2A1LT01';
	"Cip".obiekt[#nr].typObiektu :=18;
	"Cip".obiekt[#nr].inPomiarRaw := "aiC2A1LT01";
	#real := "Cip".obiekt[#nr].WartośćPomiaru;
	//
	#nr := 15;//tu wpisz nuemr obiektu
	"Cip".tor[1].zbiornikDezynfekantu.poziomAnalogowy := #nr; ;//tu przyporządkuj numer do obiektu na odpowiednim torze stacji
	;//tu wpisz nazwę
	"Cip".obiekt[#nr].nazwaObiektu := 'C2D1LT01';
	"Cip".obiekt[#nr].typObiektu := 18;
	"Cip".obiekt[#nr].inPomiarRaw := "aiC2D1LT01";
	#real := "Cip".obiekt[#nr].WartośćPomiaru;
	//
	#nr := 16;//tu wpisz nuemr obiektu
	"Cip".tor[2].zbiornikDezynfekantu.poziomAnalogowy:= #nr; ;//tu przyporządkuj numer do obiektu na odpowiednim torze stacji
	;//tu wpisz nazwę
	"Cip".obiekt[#nr].nazwaObiektu := 'C2D2LT01';
	"Cip".obiekt[#nr].typObiektu := 18;
	"Cip".obiekt[#nr].inPomiarRaw := "aiC2D2LT01";
	#real := "Cip".obiekt[#nr].WartośćPomiaru;
	//
	#nr := 17;//tu wpisz nuemr obiektu
	"Cip".tor[1].zbiornikDezynfekantu_2.poziomAnalogowy := #nr; ;//tu przyporządkuj numer do obiektu na odpowiednim torze stacji
	;//tu wpisz nazwę
	"Cip".obiekt[#nr].nazwaObiektu := 'C2D3LT01';
	"Cip".obiekt[#nr].typObiektu :=18;
	"Cip".obiekt[#nr].inPomiarRaw := "aiC2D3LT01";
	#real := "Cip".obiekt[#nr].WartośćPomiaru;
	//
	#nr := 18;//tu wpisz nuemr obiektu
	"Cip".tor[0].zbiornikŁugu.poziomAnalogowy := #nr; ;//tu przyporządkuj numer do obiektu na odpowiednim torze stacji
	;//tu wpisz nazwę
	"Cip".obiekt[#nr].nazwaObiektu := 'C2L1LT01';
	"Cip".obiekt[#nr].typObiektu := 18;
	"Cip".obiekt[#nr].inPomiarRaw := "aiC2L1LT01";
	#real := "Cip".obiekt[#nr].WartośćPomiaru;
	//
	#nr := 19;//tu wpisz nuemr obiektu
	"Cip".tor[0].zbiornikWodyWtórnej.poziomAnalogowy := #nr; ;//tu przyporządkuj numer do obiektu na odpowiednim torze stacji
	;//tu wpisz nazwę
	"Cip".obiekt[#nr].nazwaObiektu := 'C2R1LT01';
	"Cip".obiekt[#nr].typObiektu := 18;
	"Cip".obiekt[#nr].inPomiarRaw := "aiC2R1LT01";
	#real := "Cip".obiekt[#nr].WartośćPomiaru;
	//
	#nr := 20;//tu wpisz nuemr obiektu
	"Cip".tor[0].zbiornikwodyCzystej.poziomAnalogowy := #nr; ;//tu przyporządkuj numer do obiektu na odpowiednim torze stacji
	;//tu wpisz nazwę
	"Cip".obiekt[#nr].nazwaObiektu := 'C2W1LT01';
	"Cip".obiekt[#nr].typObiektu := 18;
	"Cip".obiekt[#nr].inPomiarRaw := "aiC2W1LT01";
	#real := "Cip".obiekt[#nr].WartośćPomiaru;
	
	
	////////////////////////konduktometr
	#nr := 12;//tu wpisz nuemr obiektu
	"Cip".tor[2].przewodnośćNaPowrocie := #nr; ;//tu przyporządkuj numer do obiektu na odpowiednim torze stacji
	"Cip".obiekt[#nr].nazwaObiektu := 'C212QIC01';
	"Cip".obiekt[#nr].typObiektu := 12;
	
	#REALWEJSCIE := INT_TO_REAL("aiC212QIC01");
	#real := #REALWEJSCIE;
	
	
	#aktualnyNumerReceptury := "Tor1_RecepturyStacjaMycia".numerUżywanejReceptury;
	#aktualnyKrokMycia := "Tor1_RecepturyStacjaMycia".numerKrokuMycia;
	IF "Tor1_RecepturyStacjaMycia".Receptura[#aktualnyNumerReceptury].Krok[#aktualnyKrokMycia].PM[22] = 1
	THEN
	    #real := #REALWEJSCIE /
	    (1 + (("Cip".obiekt["C212QIC01"].WartośćPomiaru -
	    "Tor1_RecepturyStacjaMycia".Receptura[#aktualnyNumerReceptury].Krok[#aktualnyKrokMycia].PM[18])
	    * "Tor1_RecepturyStacjaMycia".Receptura[#aktualnyNumerReceptury].Krok[#aktualnyKrokMycia].PM[17]) / 100);
	
	END_IF;
	
	
	"Cip".obiekt["C212QIC01"].inPomiarRaw := REAL_TO_INT(#real);
	#real := "Cip".obiekt["C212QIC01"].WartośćPomiaru;
	
	
	////////////////////////////////////////////////
	#nr := 13;//tu wpisz nuemr obiektu
	"Cip".tor[1].przewodnośćNaPowrocie := #nr; ;//tu przyporządkuj numer do obiektu na odpowiednim torze stacji
	;//tu wpisz nazwę
	"Cip".obiekt[#nr].nazwaObiektu := 'C211QIC01';
	"Cip".obiekt[#nr].typObiektu := 12;
	
	#REALWEJSCIE := INT_TO_REAL("aiC211QIC01");
	#real := #REALWEJSCIE;
	
	
	#aktualnyNumerReceptury := "Tor1_RecepturyStacjaMycia".numerUżywanejReceptury;
	#aktualnyKrokMycia := "Tor1_RecepturyStacjaMycia".numerKrokuMycia;
	IF "Tor1_RecepturyStacjaMycia".Receptura[#aktualnyNumerReceptury].Krok[#aktualnyKrokMycia].PM[22] = 1
	THEN
	    #real := #REALWEJSCIE /
	    (1 + (("Cip".obiekt["C211QIC01"].WartośćPomiaru -
	    "Tor1_RecepturyStacjaMycia".Receptura[#aktualnyNumerReceptury].Krok[#aktualnyKrokMycia].PM[18])
	    * "Tor1_RecepturyStacjaMycia".Receptura[#aktualnyNumerReceptury].Krok[#aktualnyKrokMycia].PM[17]) / 100);
	    
	END_IF;
	
	
	"Cip".obiekt["C211QIC01"].inPomiarRaw := REAL_TO_INT(#real);
	#real := "Cip".obiekt["C211QIC01"].WartośćPomiaru;
	
	
	
	
	
	
	// // //przepływomierze
	
	#nr:=106 ;//tu wpisz nuemr obiektu
	"Cip".tor[1].przepływomierzZaWymiennikiem := #nr; ;//tu przyporządkuj numer do obiektu na odpowiednim torze stacji
	"Cip".obiekt[#nr].nazwaObiektu := 'C201FT01';
	"Cip".obiekt[#nr].typObiektu := 17;
	// "Cip".obiekt[#nr].inPomiarRaw := "aiC101FT11";
	// #real:="Cip".obiekt[#nr].WartośćPomiaru;
	
	"Cip".obiekt[#nr].pomiarTymczas:="C201FT01volume";
	
	
	#nr := 107;//tu wpisz nuemr obiektu
	"Cip".tor[2].przepływomierzZaWymiennikiem := #nr; ;//tu przyporządkuj numer do obiektu na odpowiednim torze stacji
	"Cip".obiekt[#nr].nazwaObiektu := 'C202FT01';
	"Cip".obiekt[#nr].typObiektu := 17;
	// "Cip".obiekt[#nr].inPomiarRaw := "aiC101FT11";
	// #real:="Cip".obiekt[#nr].WartośćPomiaru;
	
	"Cip".obiekt[#nr].pomiarTymczas := "C202FT01volume";
	
	
	
	// ////////////////////////////////////  zawory analogowe
	// //   
	// //
	#nr:=21 ;//tu wpisz nuemr obiektu
	"Cip".tor[1].zawórParowyRegulacyjny := #nr; ;//tu przyporządkuj numer do obiektu na odpowiednim torze stacji
	"Cip".obiekt[#nr].nazwaObiektu := 'C202CV21';
	"Cip".obiekt[#nr].typObiektu := 2;
	"Cip".obiekt[#nr].inZezwolenieNaPracę := #diKSB_OK;
	"aoC201CV21" := REAL_TO_INT("Cip".obiekt[#nr].outWysterowanieUrządzenia  * 276.48);
	//
	// //
	#nr := 22;//tu wpisz nuemr obiektu
	"Cip".tor[2].zawórParowyRegulacyjny := #nr; ;//tu przyporządkuj numer do obiektu na odpowiednim torze stacji
	;//tu wpisz nazwę
	"Cip".obiekt[#nr].nazwaObiektu := 'C202CV21';
	"Cip".obiekt[#nr].typObiektu := 2;
	"Cip".obiekt[#nr].inZezwolenieNaPracę := #diKSB_OK;
	"aoC202CV21" := REAL_TO_INT("Cip".obiekt[#nr].outWysterowanieUrządzenia * 276.48);
	
END_FUNCTION

FUNCTION "Tor1.aMAIN" : Void
{ S7_Optimized_Access := 'TRUE' }
VERSION : 0.1

BEGIN
	//ponizsze FC należy napisać dla każdego urządzenia od nowa
	"Tor1.kroki"();
	"Tor1.procedury_alarmow"();
	"Tor1.procedury_obiektów"();
	"Tor1.procedury_sygnałów"();
	"Tor1_RecepturyStacjaMycia"();
	
	
	
	
	
	
	
	
	
END_FUNCTION

FUNCTION "Tor1.kroki" : Void
{ S7_Optimized_Access := 'TRUE' }
VERSION : 0.1
   VAR_TEMP 
      fdsf : Int;
      doSkasowania : Int;
      aktualnyNumerReceptury : Int;
      aktualnyKrokMycia : Int;
      sygnały_S1_czujnik_S1M1ZS02 : Bool;
   END_VAR


BEGIN
	    #aktualnyNumerReceptury := "Tor1_RecepturyStacjaMycia".numerUżywanejReceptury;
	    #aktualnyKrokMycia := "Tor1_RecepturyStacjaMycia".numerKrokuMycia;
	    "Tor1_program".program.numerKrMycia := "Tor1_RecepturyStacjaMycia".numerKrokuMycia;
	    "linia1_pompa_zezwolenie" := 1;
	    
	
	    
	    IF
	        "Tor1_hmi".button.bStop.set = 1
	        // OR "diSAFETY"=0
	    THEN
	        "Tor1_program".program.numerKroku :=7100;
	        "Tor1_hmi".button.bStop.set := 0;
	        "Tor1_hmi".button.bStart.set := 0;
	        "Tor1_hmi".button.bProdukcja.set := 0;
	        "Tor1_hmi".button.bPrzygotowanie.set := 0;
	        "Tor1_hmi".button.bPullout.set := 0;
	        "Tor1_hmi".button.bCyrkulacja.set := 0;
	        "Tor1_hmi".button.bFlux.set := 0;
	        "Tor1_hmi".button.bCip.set := 0;
	    END_IF;
	    
	    
	    "Tor1_hmi".button.bStop.kolor := BOOL_TO_INT("Tor1_hmi".button.bStop.set);
	    "Tor1_hmi".button.bStart.kolor:= BOOL_TO_INT("Tor1_hmi".button.bStart.set) ;
	    "Tor1_hmi".button.bProdukcja.kolor := BOOL_TO_INT("Tor1_hmi".button.bProdukcja.set) ;
	    "Tor1_hmi".button.bPrzygotowanie.kolor := BOOL_TO_INT("Tor1_hmi".button.bPrzygotowanie.set);
	    "Tor1_hmi".button.bPullout.kolor :=BOOL_TO_INT("Tor1_hmi".button.bPullout.set) ;
	    "Tor1_hmi".button.bCyrkulacja.kolor := BOOL_TO_INT("Tor1_hmi".button.bCyrkulacja.set);
	    "Tor1_hmi".button.bFlux.kolor := BOOL_TO_INT("Tor1_hmi".button.bFlux.set);
	    "Tor1_hmi".button.bCip.kolor :=BOOL_TO_INT("Tor1_hmi".button.bCip.set) ;
	    "Tor1_hmi".button.bPauza.kolor := BOOL_TO_INT("Tor1_hmi".button.bPauza.set AND "Clock_1Hz")*2;
	    
	
	    
	    
	    CASE "Tor1_program".program.numerKroku OF
	            
	        0: //inicjalizacja   
	            "IdźDoKroku"(inNumerKrokuDocelowy := 7100,
	                         inZadaneOpóżnienie   := 1,
	                         numerKroku           := "Tor1_program".program.numerKroku,
	                         opóźnienie           := "Tor1_program".program.opóżnienie,
	                         pauza:=  "Tor1_hmi".button.bPauza.set);
	            
	        7100://Postój
	            
	            "Cip".obiekt["Cip".tor[1].przepływomierzZaWymiennikiem].licznik1 := 0;
	            IF
	                "Tor1_hmi".button.bStart.set = 1
	            THEN
	                "IdźDoKroku"(inNumerKrokuDocelowy := 7200,
	                             inZadaneOpóżnienie   := 1,
	                             numerKroku           := "Tor1_program".program.numerKroku,
	                             opóźnienie           := "Tor1_program".program.opóżnienie,
	                             pauza:=  "Tor1_hmi".button.bPauza.set);
	                "Tor1_RecepturyStacjaMycia".numerKrokuMycia := 1;
	            END_IF;
	            
	            IF
	                "Tor1_hmi".button.bPrzygotowanie.set = 1
	            THEN
	                "IdźDoKroku"(inNumerKrokuDocelowy := 7300,
	                             inZadaneOpóżnienie   := 1,
	                             numerKroku           := "Tor1_program".program.numerKroku,
	                             opóźnienie           := "Tor1_program".program.opóżnienie,
	                             pauza:=  "Tor1_hmi".button.bPauza.set);
	                "Tor1_RecepturyStacjaMycia".numerKrokuMycia := 3;
	            END_IF;
	            
	            IF
	                "Tor1_hmi".button.bCip.set = 1
	            THEN
	                "IdźDoKroku"(inNumerKrokuDocelowy := 7400,
	                             inZadaneOpóżnienie := 1,
	                             numerKroku := "Tor1_program".program.numerKroku,
	                             opóźnienie := "Tor1_program".program.opóżnienie,
	                             pauza:=  "Tor1_hmi".button.bPauza.set);
	                "Tor1_RecepturyStacjaMycia".numerKrokuMycia := 1;
	            END_IF;
	            
	            "Tor1_program".program.zadana1 := 0;
	            "Tor1_program".program.aktualna1 := 0;
	            "Tor1_program".program.zadana2 := 0;
	            "Tor1_program".program.aktualna2 := 0;
	           
	            
	            
	            
	        7200://Zaczytanie numeru receptury (program ustawia Krok mycia =1)
	            
	            IF "Tor1_RecepturyStacjaMycia".bPokazOknoWyboruReceptury = 0 THEN
	                "Tor1_RecepturyStacjaMycia".bPokazOknoWyboruReceptury := 1;
	            END_IF;
	            IF
	                "Tor1_RecepturyStacjaMycia".klawiszUżyjTejReceptury = 1
	            THEN
	                "IdźDoKroku"(inNumerKrokuDocelowy := 7201,
	                             inZadaneOpóżnienie := 0,
	                             numerKroku := "Tor1_program".program.numerKroku,
	                             opóźnienie := "Tor1_program".program.opóżnienie,
	                             pauza := "Tor1_hmi".button.bPauza.set);
	                "Tor1_RecepturyStacjaMycia".bPokazOknoWyboruReceptury := 0;
	               
	                #doSkasowania := 1;
	                
	
	                
	                
	            END_IF;
	            "Tor1_program".program.zadana1 := 0;
	            "Tor1_program".program.aktualna1 := 0;
	            "Tor1_program".program.zadana2 := 0;
	            "Tor1_program".program.aktualna2 := 0;
	            
	            
	            #aktualnyNumerReceptury := "Tor1_RecepturyStacjaMycia".numerWyswietlanejReceptury;
	            IF "Tor1_RecepturyStacjaMycia"."klawiszReceptura-1" OR "Tor1_RecepturyStacjaMycia"."klawiszReceptura+1" THEN
	                "Tor1_hmi".bPomińŁugowanie := NOT
	                INT_TO_BOOL("Tor1_RecepturyStacjaMycia".Receptura[#aktualnyNumerReceptury].Krok[3].PM[1]);
	                "Tor1_hmi".bPomińKwasowanie := NOT
	                INT_TO_BOOL("Tor1_RecepturyStacjaMycia".Receptura[#aktualnyNumerReceptury].Krok[4].PM[1]);
	                "Tor1_hmi".bPomińDesynfekcje := NOT
	                INT_TO_BOOL("Tor1_RecepturyStacjaMycia".Receptura[#aktualnyNumerReceptury].Krok[6].PM[1]);
	            END_IF;
	         7201: //      Potwierdzenie gotowości obiektu
	             #aktualnyNumerReceptury := #aktualnyNumerReceptury;
	             #aktualnyKrokMycia := #aktualnyKrokMycia;
	             "Tor1_RecepturyStacjaMycia".Receptura[#aktualnyNumerReceptury].Krok[#aktualnyKrokMycia].PM[23]:=
	             "Tor1_RecepturyStacjaMycia".Receptura[#aktualnyNumerReceptury].Krok[#aktualnyKrokMycia].PM[23] ;
	            // jeżeli wybrano sprawdzenie czujnika
	            IF "Tor1_RecepturyStacjaMycia".Receptura[#aktualnyNumerReceptury].Krok[#aktualnyKrokMycia].PM[21] = 1
	                //sprawdzenie czujnika dla wybranego obiektu
	            THEN
	                //jezeli wybrano obiekt do mycia numer 1234
	                //
	                "CipSignals".Object[
	                REAL_TO_INT("Tor1_RecepturyStacjaMycia".Receptura[#aktualnyNumerReceptury].Krok[#aktualnyKrokMycia].PM[24])].toCip.bReadyToCip := "CipSignals".Object[0].toCip.bReadyToCip;
	                IF 
	                    // "SIG".SIG[
	                    // REAL_TO_INT("Tor1_RecepturyStacjaMycia".Receptura[#aktualnyNumerReceptury].Krok[#aktualnyKrokMycia].PM[24])]=1
	                    //i jest sygnał z czujnika
	                    //AND #sygnały_S1_czujnik_S1M1ZS02 = 1
	                   
	                    "CipSignals".Object[
	                    REAL_TO_INT("Tor1_RecepturyStacjaMycia".Receptura[#aktualnyNumerReceptury].Krok[#aktualnyKrokMycia].PM[24])].toCip.bReadyToCip=1
	                    THEN
	                    "IdźDoKroku"(inNumerKrokuDocelowy := 7202,
	                                 inZadaneOpóżnienie   := 5,
	                                 numerKroku           := "Tor1_program".program.numerKroku,
	                                 opóźnienie           := "Tor1_program".program.opóżnienie,
	                                 pauza:=  "Tor1_hmi".button.bPauza.set);
	                END_IF;
	            ELSE
	                "IdźDoKroku"(inNumerKrokuDocelowy := 7202,
	                             inZadaneOpóżnienie := 10,
	                             numerKroku := "Tor1_program".program.numerKroku,
	                             opóźnienie := "Tor1_program".program.opóżnienie,
	                             pauza := "Tor1_hmi".button.bPauza.set);
	            END_IF;
	            
